                uiBothStep := 3100;
            3100:
                IF DAS_CoreSys.MachineControl.fballocatearea.fbPulloutCv.Done THEN
                    DAS_CoreSys.MachineControl.fballocatearea.M_StopStoragePulloutAction();
                    BoxReady_2nd := TRUE;
                    uiBothStep := 9999;
                END_IF

                IF DAS_CoreSys.MachineControl.fballocatearea.fbPulloutCv.Error THEN
                    DAS_CoreSys.MachineControl.fballocatearea.M_StopStoragePulloutAction();
                    uiResumeStep := 30000;
                    uiBothStep := 3000;
                    _Abort := TRUE;
                    strStatus := 'FB_RobotRegionMove_PullOutConveyor Step 30000: Feed box timeout';


                END_IF
            9999: //Wait		
        // wait reset
        END_CASE

        // Robot Abs move
        Robot.M_StartRobotAbsMove(GetBox := Get,
                                  UseClampA := UseA,
                                  UseClampB := UseB,
                                  Area := Area,
                                  ClampA_Address := Address_A,
                                  ClampB_Address := Address_B,
                                  BoxReady_1 := BoxReady_1st,
                                  BoxReady_2 := BoxReady_2nd);

        IF Robot._DI1.Done THEN
            tonTimeOut.IN := FALSE;
            uiExecutingStep := 30080;
        END_IF

        tonTimeOut.IN := TRUE;

        IF tonTimeOut.Q = TRUE THEN
            tonTimeOut.IN := FALSE;
            strStatus 	  := 'FB_RobotRegionMove_PullOutConveyor Step 30000: Robot Move timeout';
			uiResumeStep := 30000;
            _Abort := TRUE;
        END_IF
		IF robot._DI1.Error THEN
			_Abort		 := TRUE;
			strStatus	 := CONCAT('FB_RobotRegionMove_PullOutConveyor Step 30000: ',robot.ErrMsg);
			uiResumeStep := 30000;
		END_IF

    30080: // Check robot command is clear

        Robot.M_ResetRobotAbsMove(UseA, UseB);
        DAS_CoreSys.MachineControl.fballocatearea.M_StopStoragePulloutAction();

        IF NOT Robot._DI1.Done THEN
            tonTimeOut.IN := FALSE;
            uiExecutingStep := 99000; // 
        END_IF

        tonTimeOut.IN := TRUE;

        IF tonTimeOut.Q = TRUE THEN
            strStatus := 'FB_RobotRegionMove_PullOutConveyor Step 30080: Stop Robot timeout';


            _Error := TRUE;
        END_IF

    99000: // process done
        DAS_CoreSys.MachineControl.fballocatearea.M_ReleasePulloutAccess(ControlAccess := E_RoundBeltControlAccess.FanucRobot);
        Status := 'FB_RobotRegionMove_PullOutConveyor Step 99000: Process completed';
        _Executed := TRUE;
END_CASE

IF _Executed THEN
    eState := STATE_DONE;
ELSIF _Error THEN

    eState := STATE_ERROR;
ELSIF NOT Execute THEN
    eState := STATE_RESETTING;
END_IF

IF _Abort OR Abort THEN

    eSTATE := STATE_ABORTING;
END_IF
END_METHOD

METHOD  M_STATE_RESETTING
VAR_INPUT
END_VAR
// Done := false 更改到Dormant 清除確保，上位檢查到done 後可以直接下Execute

CASE uiResettingStep OF

    0:
        tonTimeOut.IN := FALSE;
        Robot.M_ResetAllCommand();
        Robot.M_ResetRobotAbsMove(TRUE, TRUE);
        uiResettingStep := 100;
        DAS_CoreSys.MachineControl.fbStorageArea.M_ResetSlides_FeedOut();
    100:

        // DAS_CoreSys.MachineControl.fbStorageArea.M_InactivePulloutConveyorInternCtrl();
        DAS_CoreSys.MachineControl.fbAllocateArea.M_ReleasePulloutAccess(ControlAccess := E_RoundBeltControlAccess.FanucRobot);
        DAS_CoreSys.MachineControl.fbAllocateArea.M_StopStoragePulloutAction();
        uiResettingStep := 9999;
    9999:
//        Done := FALSE;
//        Busy := FALSE;
        _ResetCompleted := TRUE;
END_CASE

IF _ResetCompleted THEN
    eSTATE := STATE_DORMANT;
END_IF
END_METHOD

END_FUNCTION_BLOCK

// ---- Library/20_MachineUnits/22_AllocateArea/Service/FB_AllocateRobotNeedlingMove.TcPOU
FUNCTION_BLOCK FB_AllocateRobotNeedlingMove EXTENDS FB_ActionBasic
VAR_INPUT
    xExecute      : BOOL;
    xAbort        : BOOL;
    TimeOut  : LREAL := 30; // Unit : s
	MovingInfo	: ST_AllocateRobotNeedlingMoveInfo;
END_VAR
VAR_OUTPUT
    xAborted : BOOL;
    iErrorID : INT;
    ErrorMsg : T_MaxString;
END_VAR
VAR
    StateBehavior   : CBML.ETrigATo;
    uiCyclicStep    : UINT := 0;
    uiIndexLoop     : UINT;
	Coordinate		:st_Coordinate;
	fbExecuteEdgeDetect :FB_EdgeDetect;
END_VAR

THIS^.IBehaviourModel := StateBehavior;
StateBehavior(xExecute := xExecute,
              xAbort := xAbort OR fbExecuteEdgeDetect.xFallingEdge,
              udiTimeOut := LREAL_TO_UDINT( TimeOut*1000000),
              xDone => xDone,
              xBusy => xBusy,
              xError => xError,			  
              xAborted => xAborted);			  

			  
//Make sure that C# turns off execute to shut down the service
fbExecuteEdgeDetect(xInput :=xExecute);

//Error Msg
iErrorID := StateBehavior._model.iErrorID;
ErrorMsg := M_GetErrorMsg(xErrorID := iErrorID);

METHOD CleanupAction
VAR_INPUT
    xAbortProposed : BOOL;
    iErrorIDProposed: INT;
END_VAR
VAR_OUTPUT
    xComplete : BOOL := TRUE;
    xAbort: BOOL := xAbortProposed;
 	iErrorID : INT := iErrorIDProposed;
END_VAR
uiCyclicStep := 0;
END_METHOD

METHOD CyclicAction
VAR_INPUT
    itfTimingController : CBML.ITimingController;
END_VAR
VAR_OUTPUT
    xComplete : BOOL := TRUE;
    iErrorID : INT := 0;
END_VAR
VAR_INST
	
END_VAR

VAR
		bAxesCheck 		: BOOL;
	
	
END_VAR
xComplete := FALSE;

	IF arAxisCtrl_gb[AxisNo.Allocate_X].Admin.Axis.Status.Error OR
		arAxisCtrl_gb[AxisNo.Allocate_Y].Admin.Axis.Status.Error THEN
		iErrorID :=3;
	END_IF

CASE uiCyclicStep OF
    0:
		
			uiCyclicStep:=100;
		
		
	100:
			arAxisCtrl_gb[AxisNo.Allocate_X].PosMode.Position:=Coordinate.X;
			arAxisCtrl_gb[AxisNo.Allocate_Y].PosMode.Position:=Coordinate.Y;	
		
			IF arAxisCtrl_gb[AxisNo.Allocate_X].Admin.Axis.Status.Moving OR
			   arAxisCtrl_gb[AxisNo.Allocate_Y].Admin.Axis.Status.Moving OR
			   arAxisStatus_gb[AxisNo.Allocate_X].Admin._OpModeAck=E_AXIS_MODE.ModePosAbs OR
			   arAxisStatus_gb[AxisNo.Allocate_y].Admin._OpModeAck=E_AXIS_MODE.ModePosAbs THEN
			   uiCyclicStep:=200;
			END_IF
			
	200:
			bAxesCheck := TRUE;

		bAxesCheck := bAxesCheck AND	 arAxisStatus_gb[AxisNo.Allocate_x].Admin.CmdDone ;
		bAxesCheck := bAxesCheck AND	 arAxisStatus_gb[AxisNo.Allocate_y].Admin.CmdDone ;	
	
		IF bAxesCheck THEN
			 uiCyclicStep:=600;
		END_IF
	600:
		
		xComplete := TRUE;
END_CASE
END_METHOD

METHOD ExitAction
VAR_INPUT
    xAfterCleanup : BOOL;
    xInCopyCode : BOOL;
END_VAR
END_METHOD

METHOD PRIVATE M_CheckCommand : BOOL
VAR_INPUT
END_VAR
VAR_OUTPUT
	iErrorID	 : INT :=0 ;
END_VAR
VAR
	
END_VAR
IF MovingInfo.Box<0 OR MovingInfo.Box >1 OR MovingInfo.Clip<0 OR MovingInfo.Clip>3 OR MovingInfo.NeedleLocation<0 OR MovingInfo.NeedleLocation>49 THEN
	iErrorID :=2;
	M_CheckCommand := FALSE;
	RETURN;
END_IF

IF MovingInfo.Area = 'T' THEN
		
	FUN_GetNeedleCoordinates(uiLocation :=1 ,
							 uiBox:=MovingInfo.Box,
							 uiClip:=MovingInfo.Clip,
							 uiNeedleLocation:=MovingInfo.NeedleLocation,
							 NeedleCoordinate=>Coordinate);
	IF MovingInfo.Box = 1 AND (MovingInfo.Clip = 2 OR MovingInfo.Clip = 3) THEN
		M_CheckCommand := FALSE;
		iErrorID :=2;
		RETURN;
	END_IF
	IF MovingInfo.Box = 2 AND (MovingInfo.Clip = 0 OR MovingInfo.Clip = 1) THEN
		M_CheckCommand :=FALSE;
		iErrorID :=2;
		RETURN;
	END_IF
	
ELSIF 	

	MovingInfo.Area = 'Q' THEN
	FUN_GetNeedleCoordinates(uiLocation :=0 ,
							 uiBox:=MovingInfo.Box,
							 uiClip:=MovingInfo.Clip,
							 uiNeedleLocation:=MovingInfo.NeedleLocation,
							 NeedleCoordinate=>Coordinate);
	

ELSE
	iErrorID :=2;
	M_CheckCommand := FALSE;
	RETURN;
END_IF

M_CheckCommand:=TRUE;
END_METHOD

METHOD M_GetErrorMsg : T_MaxString
VAR_INPUT
	xErrorID: INT;
END_VAR

VAR
	
END_VAR
CASE xErrorID OF
	0:
		M_GetErrorMsg := 'No Error';
	1:
		M_GetErrorMsg := 'FB_AllocateRobotNeedlingMove ErrorID 1: Action time out';
	2:
		M_GetErrorMsg := 'FB_AllocateRobotNeedlingMove ErrorID 2: Wrong command';
	3:
		M_GetErrorMsg := 'FB_AllocateRobotNeedlingMove ErrorID 3: Servo axis error';
//	4:
//		M_GetErrorMsg := 'Axis roundbelt not ready has Error';
//	5:
//		M_GetErrorMsg := 'Cylinder not ready has Error';
//	6:
//		M_GetErrorMsg := 'Axis RoundBelt has Error';
//	7:
//		M_GetErrorMsg := 'ChargeZone_Plug has Error';
//	8:
//		M_GetErrorMsg := 'TransmitCVZone_Plug has Error';
//	9:
//		M_GetErrorMsg := 'WorkZone_Plug has Error';
//	10:
//		M_GetErrorMsg := 'WorkZone_Press has Error';
END_CASE
END_METHOD

METHOD PRIVATE M_ResetAxes : BOOL
VAR_INPUT
END_VAR
VAR
	bAxesCheck :BOOL;
END_VAR
		bAxesCheck :=TRUE;
		IF arAxisCtrl_gb[AxisNo.Allocate_X].Admin.Axis.Status.Error THEN
			arAxisCtrl_gb[AxisNo.Allocate_X].Admin.ClearError:=TRUE;			
			ELSE
			arAxisCtrl_gb[AxisNo.Allocate_X].Admin.ClearError:=FALSE;	
		END_IF
		IF arAxisCtrl_gb[AxisNo.Allocate_Y].Admin.Axis.Status.Error THEN
			arAxisCtrl_gb[AxisNo.Allocate_Y].Admin.ClearError:=TRUE;			
			ELSE
			arAxisCtrl_gb[AxisNo.Allocate_Y].Admin.ClearError:=FALSE;	
		END_IF
		bAxesCheck := bAxesCheck AND NOT arAxisCtrl_gb[AxisNo.Allocate_X].Admin.ClearError ;
		bAxesCheck := bAxesCheck AND NOT arAxisCtrl_gb[AxisNo.Allocate_X].Admin.ClearError ;
		
		M_ResetAxes := bAxesCheck;
END_METHOD

METHOD ResetAction
VAR_OUTPUT
    xComplete : BOOL := TRUE;
END_VAR
uiCyclicStep := 0;
END_METHOD

METHOD StartAction
VAR_OUTPUT
    xComplete : BOOL := TRUE;
	iErrorID : INT := 0;
END_VAR
xComplete := FALSE;
uiCyclicStep := 0;

IF M_CheckCommand(iErrorID=>iErrorID) AND M_ResetAxes() THEN
	xComplete := TRUE;
END_IF
END_METHOD

END_FUNCTION_BLOCK

// ---- Library/20_MachineUnits/21_StorageArea/FB_StorageArea.TcPOU
FUNCTION_BLOCK FB_StorageArea EXTENDS FB_ModeBase_V2 IMPLEMENTS I_UnitState
VAR_INPUT
    FanucRobot : REFERENCE TO FB_FanucRobot_Basic_V2;
    Service    : REFERENCE TO ST_StorageService;

    Cylinder : REFERENCE TO UNI_CylinderList;
    Motor    : REFERENCE TO UNI_MotorList;

    Input            : REFERENCE TO ST_InputTable;
    OutPut           : REFERENCE TO ST_OutputTable;
    Reset            : REFERENCE TO BOOL;
	Stop :  REFERENCE TO BOOL;
	bStopMem :  REFERENCE TO BOOL;
    WheelhouseSensor : REFERENCE TO UNI_HMI_WheelHouseInput;
    CurrentData      : ST_SetupPara;
END_VAR
VAR_OUTPUT
	RobotResetCMD :BOOL;
	Homed : BOOL;
END_VAR
VAR
	Abort	:BOOL;

	// 連動暫停 - 任一 Service 錯誤時暫停所有其他 Service
	_bAnyServiceError : BOOL;

    // Service
    //fbFeedInEmptyBoxWithRobot           : FB_FeedInEmptyBoxWithRobot;
	fbFeedInEmptyBoxWithRobot           : FB_FeedInEmptyBoxWithRobot_V4;			//Edited by Gamin in 2025//11/24
    //fbReloadRoundBeltBoxWithRobot       : FB_ReloadRoundBeltBoxWithRobot;
	fbReloadRoundBeltBoxWithRobot       : FB_ReloadRoundBeltBoxWithRobot_V2;		//Edited by Gamin in 2025//11/24
    fbRobotRegionMove_AllocatedConveyor : FB_RobotRegionMove_AllocatedConveyor;
    fbRobotRegionMove_BufferArea        : FB_RobotRegionMove_BufferArea;
    //fbRobotRegionMove_FeedInConveyor    : FB_RobotRegionMove_FeedInConveyor;
	fbRobotRegionMove_FeedInConveyor    : FB_RobotRegionMove_FeedInConveyor_V2;		//Edited by Gamin in 2025//11/24
    fbRobotRegionMove_PullOutConveyor   : FB_RobotRegionMove_PullOutConveyor;
    fbRobotRegionMove_RoundBelt         : FB_RobotRegionMove_RoundBelt;
    //fbRobotAbsMove                      : FB_RobotAbsMove;
	fbRobotAbsMove                      : FB_RobotAbsMove_V2;
    //fbWareHouseWithRobotMove            : FB_WareHouseWithRobotMove;
    fbWareHouseWithRobotMove             : FB_WareHouseWithRobotMove_V3;		//Edited by Gamin in 2025//11/24
	fbFeedInRoundBeltBoxToWareHouse 	 : FB_FeedInRoundBeltBoxToWareHouse;
	fbWareHouseInnerPickToRoundBelt 	 : FB_WareHouseInnerPickToRoundBelt;
	fbWareHouseInnerPickToRoundBeltBatch : FB_WareHouseInnerPickToRoundBeltBatch;
	fbFeedInRoundBeltBoxBatch			 : FB_FeedInRoundBeltBoxBatch;
	fbRobotSelfHoming					 : FB_RobotSelfHoming;
	
	fbStorageHoming 					: FB_StorageHoming;
	//UpCV
    _fbDaimeterMovement   			: FB_DiameterMovement; //UpCV Internal use
    fbUpperFeedInConveyor 			: FB_UpperFeedInConveyor;
	bUpperCV_ServiceDone			: BOOL;					// 偵測上層輸送帶是否做完
	fbAddBoxes                      : FB_AddBoxes_v2;
	fbBoxSupplyCtrl					: FB_BoxSupplyCtrl_v1;
    RackState                       : E_RackState;
    
    // Pullout
    fbPullOutConveyorAction         : FB_PullOutConveyorAction;
    AutoPullout_Ctrl                : ST_AutoPullOutConveyorCommand;
    AutoPullout_Status              : ST_AutoPullOutConveyorSatus;
    AutoPullout_Info                : ST_PullOutConveyorInfo;
    bPulloutConveyorInternCtrl      : BOOL := FALSE;
    AutoMode_PulloutConveyor_Intern : ST_AutoPullOutConveyor; // Pullout conveyor inter
    

    // Robot abs move
    RobotAbsMoveAuto_Ctrl   : st_RobotAbsMove_Ctrl;
    RobotAbsMoveAuto_Status : st_RobotAbsMove_Status;
    RobotAbsMoveAuto_Info   : st_AutoSixAxisAbsMoveParameter;
    // Warehouse
	fbWarehouse           : FB_WareHouse;
    //========= Auto Mode Robot Warehouse Move =================
    RobotWarehouseMoveAuto_Ctrl   : st_RobotWarehouseMove_Ctrl;
    RobotWarehouseMoveAuto_Status : st_RobotWarehouseMove_Status;

    _RobotWarehouseMoveAuto_Ctrl   : st_RobotWarehouseMove_Ctrl;
    _RobotWarehouseMoveAuto_Status : st_RobotWarehouseMove_Status;

    RobotWarehouseMoveAuto_internal_Ctrl   : st_RobotWarehouseMove_Ctrl;
    RobotWarehouseMoveAuto_internal_Status : st_RobotWarehouseMove_Status;
    bWarehouseMoveInternalAccess           : BOOL := FALSE;
	// Storage homing
	StorageHoming_Execute : BOOL;
	StorageHoming_Reset : BOOL;
	StorageHoming_Abort : BOOL;
	StorageHoming_Busy : BOOL;
	StorageHoming_Done : BOOL;
	StorageHoming_Error : BOOL;
	
	// Reboot Modbus devices
	fbRebootModbusDevice		: FB_RebootModbusDevice;
END_VAR

SUPER^();

IF __ISVALIDREF(PackTag) THEN
    eModeCommand := PackTag.Command.UnitMode;
    eStateCommand := PackTag.Command.CntrlCmd;
ELSE
    RETURN;
END_IF

ACTION A00_Service:
// ============================================================================
// 連動暫停邏輯 - 任一 Service 錯誤時，暫停所有其他 Service
// ============================================================================
//_bAnyServiceError :=
//	service.AutoMode_FeedInEmptyBoxWithRobot.Status.Error OR
//	service.AutoMode_RobotRegionMove_BufferArea.Status.Error OR
//	service.AutoMode_UpperFeedInConveyor.Status.Error OR
//	service.AutoMode_AddBoxes.Status.Error OR
//	service.AutoMode_RobotRegionMove_FeedInConveyor.Status.Error OR
//	service.AutoMode_RobotRegionMove_AllocatedConveyor.Status.Error OR
//	service.AutoMode_RobotRegionMove_PullOutConveyor.Status.Error OR
//	service.AutoMode_RobotAbsMove.HandShake.Error OR
//	service.AutoMode_RobotRegionMove_RoundBelt.Status.Error OR
//	service.AutoMode_ReloadRoundBeltBoxWithRobot.Status.Error OR
//	service.AutoMode_WarehouseMotoWithRobotMove.HandShake.Error OR
//	AutoPullout_Status.Error;

fbFeedInEmptyBoxWithRobot(Execute    := service.AutoMode_FeedInEmptyBoxWithRobot.Command.Execute,
                          Abort      := service.AutoMode_FeedInEmptyBoxWithRobot.Command.Abort OR THIS^.Abort OR _bAnyServiceError,
                          Reset      := service.AutoMode_FeedInEmptyBoxWithRobot.Command.Reset,
                          ObjectName := 'FeedInEmptyBox with robot',
                          Busy       => service.AutoMode_FeedInEmptyBoxWithRobot.Status.Busy,
                          Done       => service.AutoMode_FeedInEmptyBoxWithRobot.Status.Done,
                          Aborted    =>,
                          Error      => service.AutoMode_FeedInEmptyBoxWithRobot.Status.Error,
                          ErrorID    =>,
                          Status     => service.AutoMode_FeedInEmptyBoxWithRobot.Status.Status,
                          UniqueErrorCode   =>,
                          Robot      := FanucRobot,
                          WareHouse  := fbWarehouse,
                          Input      := Input,
                          DiffSizeCV := Motor.List.TransmitDifferentSideCV,
						  SameSizeCV := Motor.List.TransmitSameSideCV,
                          Info := Service.AutoMode_FeedInEmptyBoxWithRobot.Info,
                          Pause := bStopMem,
                          Stop := bStopMem,
						  AClampMoveDone=>service.AutoMode_FeedInEmptyBoxWithRobot.AClampMoveDone,
						  BClampMoveDone=>service.AutoMode_FeedInEmptyBoxWithRobot.BClampMoveDone);

fbRobotRegionMove_BufferArea(Execute	:= Service.AutoMode_RobotRegionMove_BufferArea.Command.Execute,
                             Abort 		:= Service.AutoMode_RobotRegionMove_BufferArea.Command.Abort OR THIS^.Abort OR _bAnyServiceError,
                             Reset 		:= Service.AutoMode_RobotRegionMove_BufferArea.Command.Reset,
                             ObjectName	:= 'RobotRegionMove_BufferArea',
                             Busy    => Service.AutoMode_RobotRegionMove_BufferArea.Status.Busy,
                             Done    => Service.AutoMode_RobotRegionMove_BufferArea.Status.Done,
                             Aborted =>,
                             Error   => Service.AutoMode_RobotRegionMove_BufferArea.Status.Error,
                             ErrorID =>,
                             Status  => Service.AutoMode_RobotRegionMove_BufferArea.Status.Status,
							 UniqueErrorCode	=>,
                             Robot 	:= FanucRobot,
                             Info 	:= Service.AutoMode_RobotRegionMove_BufferArea.Info,
                             Stop 	:= bStopMem);

fbPullOutConveyorAction(Execute          := (*AutoPullout_Ctrl.Execute*) ,
                        Abort            := AutoPullout_Ctrl.Abort OR THIS^.Abort OR _bAnyServiceError,
                        Reset            := AutoPullout_Ctrl.Reset,
                        ObjectName       := 'fbPullOutConveyorAction',
                        Busy             => AutoPullout_Status.Busy,
                        Done             => AutoPullout_Status.Done,
                        Aborted          =>,
                        Error            => AutoPullout_Status.Error,
                        ErrorID          =>,
                        Status           => AutoPullout_Status.Status,
                        UniqueErrorCode  =>,
                        FixCylinderA1    := Cylinder.List.fbPullOutCV_AsidePress1,
                        FixCylinderA2    := Cylinder.List.fbPullOutCV_AsidePress2,
                        FixCylinderB1    := Cylinder.List.fbPullOutCV_BsidePress1,
                        FixCylinderB2    := Cylinder.List.fbPullOutCV_BsidePress2,
                        BarrierCylinderA := Cylinder.List.fbPullOutCV_AsideBlock,
                        BarrierCylinderB := Cylinder.List.fbPullOutCV_BsideBlock,
                        ConveyorMotorA   := Motor.List.PullOutCV_A,
                        ConveyorMotorB   := Motor.List.PullOutCV_B,
                        INPUT            := INPUT,
                        PullOutInfo      := AutoPullout_Info);

fbUpperFeedInConveyor(Execute             := Service.AutoMode_UpperFeedInConveyor.Command.Execute,
                      Abort               := Service.AutoMode_UpperFeedInConveyor.Command.Abort OR THIS^.Abort OR _bAnyServiceError,
                      Reset               := Service.AutoMode_UpperFeedInConveyor.Command.Reset,
                      ObjectName          := 'Storage_UpperFeedInConveyor',
                      Busy                => Service.AutoMode_UpperFeedInConveyor.Status.Busy,
                      Done                => Service.AutoMode_UpperFeedInConveyor.Status.Done,
                      Aborted             =>,
                      Error               => Service.AutoMode_UpperFeedInConveyor.Status.Error,
                      ErrorID             =>,
                      Status              =>,
                      UniqueErrorCode     =>,
                      _fbDiameterMovement := THIS^._fbDaimeterMovement,
                      Cylinder            := Cylinder,
                      Motor               := Motor,
                      Input               := Input,
                      OutPut              := OutPut,
                      Info                := Service.AutoMode_UpperFeedInConveyor.Info,
                      AddingBox           :=,
                      FeedBack            => Service.AutoMode_UpperFeedInConveyor.FeedBack,
					  _bForceUpperCV_Use  =>	,
					  Pause 			  := bStopMem,
					  RobotService_CheckUPCVServicedone =>bUpperCV_ServiceDone);

_fbDaimeterMovement(Execute         :=,
                    Abort           := _bAnyServiceError,
                    Reset           :=,
                    ObjectName      :=,
                    Busy            =>,
                    Done            =>,
                    Aborted         =>,
                    Error           =>,
                    ErrorID         =>,
                    Status          =>,
                    UniqueErrorCode =>,
                    bContinue       :=,
                    Cylinder        := Cylinder,
                    PickDone        =>);

fbWarehouse(Motors           := Motor,
            WheelhouseSensor := WheelhouseSensor);

fbAddBoxes(Execute                   := Service.AutoMode_AddBoxes.Command.Execute,
           Abort                     := Service.AutoMode_AddBoxes.Command.Abort OR THIS^.Abort OR _bAnyServiceError,
           Reset                     := Service.AutoMode_AddBoxes.Command.Reset,
           ObjectName                := 'Storage_AddBoxes',
           Busy                      => Service.AutoMode_AddBoxes.Status.Busy,
           Done                      => Service.AutoMode_AddBoxes.Status.Done,
           Aborted                   =>,
           Error                     => Service.AutoMode_AddBoxes.Status.Error,
           ErrorID                   =>,
           Status                    =>,
           UniqueErrorCode           =>,
           Cylinder                  := Cylinder,
           Motor                     := Motor,
           Input                     := Input,
           OutPut                    := OutPut,
           CurrentData               := CurrentData,
           ERackState                := RackState,
           bClearInterventionRequest :=,
           InterventionRequest       => Service.AutoMode_AddBoxes.Status.InterventionRequest,
           FeedingBoxes              => Service.AutoMode_AddBoxes.Status.FeedingBoxes,
			_bForceUpperCV_Use 		:= fbUpperFeedInConveyor._bForceUpperCV_Use);

fbBoxSupplyCtrl(Execute           := TRUE,
                Abort             :=THIS^.Abort OR _bAnyServiceError,
                Reset             :=reset,
                ObjectName        :=,
                Busy              =>,
                Done              =>,
                Aborted           =>,
                Error             =>,
                ErrorID           =>,
                Status            =>,
                UniqueErrorCode   =>,
                Cylinder          := Cylinder,
                Motor             := Motor,
                CurrentData       := CurrentData,
                Input             := Input,
                Output            := OutPut,
                StroageRegionMode := eModeCurrent,
                bAddsBoxRequest   := Service.AutoMode_AddBoxes.Status.InterventionRequest,
                AddBoxes_Status   := Service.AutoMode_AddBoxes.Status,
                AddBoxes_Ctrl     := Service.AutoMode_AddBoxes.Command,
				AxisRackMotorBTNHomeRequest=>,
                RackState         => RackState,
				fbstorageHome := fbStorageHoming);

fbRobotRegionMove_FeedInConveyor(Execute 	:= Service.AutoMode_RobotRegionMove_FeedInConveyor.Command.Execute,
                                 Abort 		:= Service.AutoMode_RobotRegionMove_FeedInConveyor.Command.Abort OR THIS^.Abort OR _bAnyServiceError,
                                 Reset      := Service.AutoMode_RobotRegionMove_FeedInConveyor.Command.Reset,
                                 ObjectName := 'Storage Robot FeedIn CV',
                                 Busy       => Service.AutoMode_RobotRegionMove_FeedInConveyor.Status.Busy,
                                 Done 		=> Service.AutoMode_RobotRegionMove_FeedInConveyor.Status.Done,
                                 Aborted	=>,
                                 Error   	=> Service.AutoMode_RobotRegionMove_FeedInConveyor.Status.Error,
                                 ErrorID 	=>,
                                 Status  	=> Service.AutoMode_RobotRegionMove_FeedInConveyor.Status.Status,
                                 UniqueErrorCode =>,
                                 Robot           := FanucRobot,
                                 LowerConveyor   := Motor.List.LowCV,
                                 Input           := Input,
                                 //								 F1SensorOfUpperConveyor :=Input.bUpCV_BoxArrived_Sensor,
                                 //								 Input.bUpCV_Block1Detect_Sensor := Input.bUpCV_Block1Detect_Sensor ,
                                 Info := Service.AutoMode_RobotRegionMove_FeedInConveyor.Info,
                                 Stop :=bStopMem,
								 bCheckUpperCV_ServiceDone :=	bUpperCV_ServiceDone);

fbRobotRegionMove_AllocatedConveyor(Execute 	:= Service.AutoMode_RobotRegionMove_AllocatedConveyor.Command.Execute,
                                    Abort 		:= Service.AutoMode_RobotRegionMove_AllocatedConveyor.Command.Abort OR THIS^.Abort OR _bAnyServiceError,
                                    Reset  		:= Service.AutoMode_RobotRegionMove_AllocatedConveyor.Command.Reset,
                                    ObjectName 	:= ' Storage Robot Transmit CV',
                                    Busy       	=> Service.AutoMode_RobotRegionMove_AllocatedConveyor.Status.Busy,
                                    Done 		=> Service.AutoMode_RobotRegionMove_AllocatedConveyor.Status.Done,
                                    Aborted 	=>,
                                    Error   	=> Service.AutoMode_RobotRegionMove_AllocatedConveyor.Status.Error,
                                    ErrorID 	=>,
                                    Status  	=> Service.AutoMode_RobotRegionMove_AllocatedConveyor.Status.Status,
                                    UniqueErrorCode =>,
                                    Robot           := FanucRobot,
                                    DifferenceCV    := Motor.List.TransmitDifferentSideCV,
                                    SamesizeCV      := Motor.List.TransmitSameSideCV,
                                    cylinder        := Cylinder,
                                    //	SameSizeFullSensor:= , 
                                    Input := Input,
                                    Info := service.AutoMode_RobotRegionMove_AllocatedConveyor.Info,
                                    Stop :=bStopMem);


fbRobotRegionMove_PullOutConveyor(Execute 	:=Service.AutoMode_RobotRegionMove_PullOutConveyor.Command.Execute,
                                  Abort 	:=Service.AutoMode_RobotRegionMove_PullOutConveyor.Command.Abort OR THIS^.Abort OR _bAnyServiceError,
                                  Reset     := Service.AutoMode_RobotRegionMove_PullOutConveyor.Command.Reset,
                                  ObjectName:= 'Storage Robot PulloutCV',
                                  Busy      => Service.AutoMode_RobotRegionMove_PullOutConveyor.Status.Busy,
                                  Done 		=> Service.AutoMode_RobotRegionMove_PullOutConveyor.Status.Done,
                                  Aborted 	=>,
                                  Error   	=> Service.AutoMode_RobotRegionMove_PullOutConveyor.Status.Error,
                                  ErrorID 	=>,
                                  Status  	=> Service.AutoMode_RobotRegionMove_PullOutConveyor.Status.Status,
                                  UniqueErrorCode =>,
                                  Robot           := FanucRobot,
                                  PullOutConveyor := fbPullOutConveyorAction,
                                  Info := Service.AutoMode_RobotRegionMove_PullOutConveyor.Info,
                                  Stop :=bStopMem);

fbRobotAbsMove(Execute         := Service.AutoMode_RobotAbsMove.HandShake.Execute,
               Abort           := THIS^.Abort OR _bAnyServiceError,
               Reset           := Service.AutoMode_RobotAbsMove.HandShake.Reset,
               ObjectName      := 'Storage robot abs move',
               Busy            => Service.AutoMode_RobotAbsMove.HandShake.Busy,
               Done            => Service.AutoMode_RobotAbsMove.HandShake.Done,
               Aborted         =>,
               Error           => Service.AutoMode_RobotAbsMove.HandShake.Error,
               ErrorID         =>,
               Status          =>,
               UniqueErrorCode =>,
               Robot           := FanucRobot,
               LowerConveyor   := Motor.List.LowCV,
               Info            := Service.AutoMode_RobotAbsMove,
               Input 		:= Input,
               Stop :=bStopMem,
			   	Output:=OutPut,
				Cylinder:= Cylinder,
				AClampMoveDone=>Service.AutoMode_RobotAbsMove.AClampMoveDone,
				BClampMoveDone=>Service.AutoMode_RobotAbsMove.BClampMoveDone,
				bCheckUpperCV_ServiceDone :=bUpperCV_ServiceDone);

fbRobotRegionMove_RoundBelt(Execute := Service.AutoMode_RobotRegionMove_RoundBelt.Command.Execute,
                            Abort   := THIS^.Abort OR _bAnyServiceError,
                            Reset   := Service.AutoMode_RobotRegionMove_RoundBelt.Command.Reset,
                            ObjectName:= 'Storage robot  RegionMove roundbelt',
                            Busy    => Service.AutoMode_RobotRegionMove_RoundBelt.Status.Busy,
                            Done    => Service.AutoMode_RobotRegionMove_RoundBelt.Status.Done,
                            Aborted =>,
                            Error   => Service.AutoMode_RobotRegionMove_RoundBelt.Status.Error,
                            ErrorID =>,
                            Status 	=> Service.AutoMode_RobotRegionMove_RoundBelt.Status.Status,
                            UniqueErrorCode =>,
                            Robot 		:= FanucRobot,
                            RoundBelt 	:= DAS_CoreSys.MachineControl.fbAllocateArea.RoundBeltControl,
							Input 		:= Input,
                            Info 		:= Service.AutoMode_RobotRegionMove_RoundBelt.Info,
                            Stop 		:=bStopMem);

fbReloadRoundBeltBoxWithRobot(Execute	:= Service.AutoMode_ReloadRoundBeltBoxWithRobot.Command.Execute,
                              Abort 	:= THIS^.Abort OR _bAnyServiceError,
                              Reset 	:= Service.AutoMode_ReloadRoundBeltBoxWithRobot.Command.Reset,
                              ObjectName:= 'Storage robot reload roundbelt',
                              Busy    => Service.AutoMode_ReloadRoundBeltBoxWithRobot.Status.Busy,
                              Done    => Service.AutoMode_ReloadRoundBeltBoxWithRobot.Status.Done,
                              Aborted =>,
                              Error   => Service.AutoMode_ReloadRoundBeltBoxWithRobot.Status.Error,
                              ErrorID =>,
                              Status  => Service.AutoMode_ReloadRoundBeltBoxWithRobot.Status.Status,
                              UniqueErrorCode =>,
                              Robot 	:= FanucRobot,
                              RoundBelt := DAS_CoreSys.MachineControl.fbAllocateArea.RoundBeltControl,
                              WareHouse := fbWarehouse,
                              Input 	:= Input,
                              Info 		:= Service.AutoMode_ReloadRoundBeltBoxWithRobot.Info,
                              Stop 		:= bStopMem,
							  AClampMoveDone=>Service.AutoMode_ReloadRoundBeltBoxWithRobot.AClampMoveDone,
							  BClampMoveDone=>Service.AutoMode_ReloadRoundBeltBoxWithRobot.BClampMoveDone);
							  
fbWareHouseInnerPickToRoundBelt(Execute	:= Service.AutoMode_WareHouseInnerPickToRoundBelt.Command.Execute,
                                Abort 	:= THIS^.Abort OR _bAnyServiceError,
                                Reset 	:= Service.AutoMode_WareHouseInnerPickToRoundBelt.Command.Reset,
                                ObjectName:= 'Warehouse inner pick to roundbelt',
                                Busy    => Service.AutoMode_WareHouseInnerPickToRoundBelt.Status.Busy,
                                Done    => Service.AutoMode_WareHouseInnerPickToRoundBelt.Status.Done,
                                Aborted =>,
                                Error   => Service.AutoMode_WareHouseInnerPickToRoundBelt.Status.Error,
                                ErrorID =>,
                                Status  => Service.AutoMode_WareHouseInnerPickToRoundBelt.Status.Status,
                                UniqueErrorCode =>,
                                Robot 	:= FanucRobot,
                                RoundBelt := DAS_CoreSys.MachineControl.fbAllocateArea.RoundBeltControl,
                                WareHouse := fbWarehouse,
                                Input 	:= Input,
                                Info 	:= Service.AutoMode_WareHouseInnerPickToRoundBelt.Info,
                                Stop 	:= bStopMem,
                                ReadComplete := Service.AutoMode_WareHouseInnerPickToRoundBelt.ReadComplete,
                                ActionRecords=>Service.AutoMode_WareHouseInnerPickToRoundBelt.ActionRecords,
                                ActionIndex=>Service.AutoMode_WareHouseInnerPickToRoundBelt.ActionIndex,
                                FeedBack=>Service.AutoMode_WareHouseInnerPickToRoundBelt.FeedBack);
fbWareHouseInnerPickToRoundBeltBatch(
                                Abort 	:= THIS^.Abort OR _bAnyServiceError,
                                ObjectName:= 'Warehouse inner pick batch',
                                Robot 	:= FanucRobot,
                                RoundBelt := DAS_CoreSys.MachineControl.fbAllocateArea.RoundBeltControl,
                                WareHouse := fbWarehouse,
                                Input 	:= Input,
                                BatchInfo := Service.AutoMode_WareHouseInnerPickToRoundBeltBatch,
                                Stop 	:= bStopMem);
// 圓帶回倉/PullOut 批次服務
fbFeedInRoundBeltBoxBatch(
                                Abort 	:= THIS^.Abort OR _bAnyServiceError,
                                ObjectName:= 'FeedIn round belt box batch',
                                Robot 	:= FanucRobot,
                                RoundBelt := DAS_CoreSys.MachineControl.fbAllocateArea.RoundBeltControl,
                                WareHouse := fbWarehouse,
                                Input 	:= Input,
                                BatchInfo := Service.AutoMode_FeedInRoundBeltBoxBatch,
                                Stop 	:= bStopMem);
								
//============================ Auto Mode Robot Warehouse Move =============================
IF NOT bWarehouseMoveInternalAccess THEN
    _RobotWarehouseMoveAuto_Ctrl := RobotWarehouseMoveAuto_Ctrl;
    RobotWarehouseMoveAuto_Status := _RobotWarehouseMoveAuto_Status;
ELSE
    _RobotWarehouseMoveAuto_Ctrl := RobotWarehouseMoveAuto_internal_Ctrl;
    RobotWarehouseMoveAuto_internal_Status := _RobotWarehouseMoveAuto_Status;
END_IF

(*M_RobotWarehouseMove(
        bExecute  := Service.AutoMode_RobotWarehouseMove.HandShake.Execute,
        bReset    := Service.AutoMode_RobotWarehouseMove.HandShake.Reset,
        bAbort    := FALSE,
        bOccupied := FALSE,
        eMode     := E_MachineMode.Auto,
        bBusy     => Service.AutoMode_RobotWarehouseMove.HandShake.Busy,
        bDone     => Service.AutoMode_RobotWarehouseMove.HandShake.Done,
        bError    => Service.AutoMode_RobotWarehouseMove.HandShake.Error);*)
fbWareHouseWithRobotMove(
	Execute:= Service.AutoMode_WarehouseMotoWithRobotMove.HandShake.Execute,
	Abort:= THIS^.Abort OR _bAnyServiceError,
	Reset:= Service.AutoMode_WarehouseMotoWithRobotMove.HandShake.Reset,
	ObjectName:= 'storage Robot Warehouse move', 
	Busy=> Service.AutoMode_WarehouseMotoWithRobotMove.HandShake.Busy, 
	Done=> Service.AutoMode_WarehouseMotoWithRobotMove.HandShake.Done, 
	Aborted=> , 
	Error=> Service.AutoMode_WarehouseMotoWithRobotMove.HandShake.Error, 
	ErrorID=> , 
	Status=> , 
	UniqueErrorCode=> , 
	Robot:= FanucRobot, 
	WareHouse:= fbWarehouse, 
	Info:= Service.AutoMode_WarehouseMotoWithRobotMove, 
	Stop:= bStopMem,
	AClampMoveDone=> Service.AutoMode_WarehouseMotoWithRobotMove.AClampMoveDone,
	BClampMoveDone=> Service.AutoMode_WarehouseMotoWithRobotMove.BClampMoveDone,
	WarehouseStatus := WheelhouseSensor.List);
	
fbStorageHoming(
	xDone=> ,
	xBusy=> ,
	xError=> ,
	xExecute:= ,
	xAbort:= THIS^.Abort OR _bAnyServiceError,
	Cylinder:= Cylinder, 
	Motor:= Motor, 
	FanucRobot:= FanucRobot,
	Homed := Homed,
	xAborted=> , 
	iErrorID=> , 
	ErrorMsg=> , 
	RobotResetCMD=> RobotResetCMD,
	RackMotorHomeRequest=>,
	Input := Input,
	Service := Service,
	Output :=OutPut);
	
fbRebootModbusDevice(
	xDone=> Service.RebootModbusDevices.Status.Done, 
	xBusy=> Service.RebootModbusDevices.Status.Busy, 
	xError=> Service.RebootModbusDevices.Status.Error, 
	xExecute:= Service.RebootModbusDevices.Command.Execute, 
	xAbort:= Service.RebootModbusDevices.Command.Abort, 
	OutPut:= OutPut, 
	OffDelayTime:= Service.RebootModbusDevices.OffDelayTime, 
	OnDelayTime:= Service.RebootModbusDevices.OnDelayTime, 
	xAborted=> , 
	iErrorID=> , 
	ErrorMsg=> );
	
fbFeedInRoundBeltBoxToWareHouse(
	Execute:= Service.AutoMode_FeedInRoundBeltBoxToWareHouse.Command.Execute, 
	Abort:= , 
	Reset:= Service.AutoMode_FeedInRoundBeltBoxToWareHouse.Command.Reset, 
	Pause:= , 
	ObjectName:= , 
	Busy=> Service.AutoMode_FeedInRoundBeltBoxToWareHouse.Status.Busy, 
	Done=> Service.AutoMode_FeedInRoundBeltBoxToWareHouse.Status.Done, 
	Aborted=> , 
	Error=> Service.AutoMode_FeedInRoundBeltBoxToWareHouse.Status.Error, 
	Paused=> , 
	ErrorID=> , 
	Status=> Service.AutoMode_FeedInRoundBeltBoxToWareHouse.Status.Status, 
	UniqueErrorCode=> , 
	Robot:= FanucRobot, 
	RoundBelt:= DAS_CoreSys.MachineControl.fbAllocateArea.RoundBeltControl, 
	WareHouse:= fbWarehouse, 
	Input:= Input, 
	Info:= Service.AutoMode_FeedInRoundBeltBoxToWareHouse.Info, 
	Stop:= bStopMem, 
	AClampMoveDone=> Service.AutoMode_FeedInRoundBeltBoxToWareHouse.AClampMoveDone, 
	BClampMoveDone=> Service.AutoMode_FeedInRoundBeltBoxToWareHouse.BClampMoveDone);
	
fbRobotSelfHoming(
	Execute:= Service.AutoMode_RobotSelfHoming.Command.Execute, 
	Abort:= , 
	Reset:= Service.AutoMode_RobotSelfHoming.Command.Reset, 
	Pause:= bStopMem, 
	ObjectName:= 'FB_RobotSelfHoming', 
	Busy=> Service.AutoMode_RobotSelfHoming.Status.Busy, 
	Done=> Service.AutoMode_RobotSelfHoming.Status.Done, 
	Aborted=> , 
	Error=> Service.AutoMode_RobotSelfHoming.Status.Error, 
	Paused=> , 
	ErrorID=> , 
	Status=> Service.AutoMode_RobotSelfHoming.Status.Status, 
	UniqueErrorCode=> , 
	FanucRobot:= FanucRobot, 
	Input:= Input, 
	Output:= OutPut, 
	Motor:= Motor, 
	BypassFeedOutToNGCV:= Service.AutoMode_RobotSelfHoming.BypassFeedOutToNGCV);
END_ACTION

METHOD M_Aborted
Abort:=FALSE;
M_StopHoming();
M_StateComplete();
END_METHOD

METHOD M_AbortHoming
VAR_INPUT
END_VAR
StorageHoming_Abort := TRUE;
END_METHOD

METHOD M_Aborting
Abort := TRUE;
M_StateComplete();
END_METHOD

METHOD M_ActivePulloutConveyorInternCtrl : BOOL
VAR_INPUT
END_VAR
bPulloutConveyorInternCtrl := TRUE;

M_ActivePulloutConveyorInternCtrl := TRUE; // Method end
END_METHOD

METHOD M_ActivePulloutConveyorInternCtrl_1 : BOOL
VAR_INPUT
END_VAR
bPulloutConveyorInternCtrl := TRUE;

M_ActivePulloutConveyorInternCtrl_1 := TRUE; // Method end
END_METHOD

METHOD M_AutoPullOutConveyorActive : BOOL
VAR_INPUT
END_VAR
IF eModeCurrent = E_UnitMode.AUTO AND NOT bPulloutConveyorInternCtrl THEN
    // GVL -> AutoSimpleAllocate_Ctrl
    AutoPullout_Ctrl.Execute := service.AutoMode_PullOutConveyor.Command.Execute;
    AutoPullout_Ctrl.Abort   := service.AutoMode_PullOutConveyor.Command.Abort;
    AutoPullout_Ctrl.Reset   := service.AutoMode_PullOutConveyor.Command.Reset OR Reset;
	M_LoadingPullOutConveyorData();
ELSIF eModeCurrent = E_UnitMode.AUTO AND bPulloutConveyorInternCtrl THEN
    AutoPullout_Ctrl.Execute := AutoMode_PulloutConveyor_Intern.Command.Execute;
    AutoPullout_Ctrl.Abort   := AutoMode_PulloutConveyor_Intern.Command.Abort;
    AutoPullout_Ctrl.Reset   := AutoMode_PulloutConveyor_Intern.Command.Reset OR Reset;
	M_LoadingPullOutConveyorData();
ELSE
    AutoPullout_Ctrl.Execute := FALSE;
    AutoPullout_Ctrl.Abort   := FALSE;
    AutoPullout_Ctrl.Reset   := FALSE;
END_IF

// AutoSimpleAllocate_Status - > GVL
service.AutoMode_PullOutConveyor.Status.Busy := AutoPullout_Status.Busy;
service.AutoMode_PullOutConveyor.Status.Done := AutoPullout_Status.Done;
service.AutoMode_PullOutConveyor.Status.Error:= AutoPullout_Status.Error;
AutoMode_PulloutConveyor_Intern.Status.Busy := AutoPullout_Status.Busy;
AutoMode_PulloutConveyor_Intern.Status.Done:= AutoPullout_Status.Done;
AutoMode_PulloutConveyor_Intern.Status.Error:= AutoPullout_Status.Error;
END_METHOD

METHOD M_Clearing
M_StateComplete();
END_METHOD

METHOD M_Complete
M_StateComplete();
END_METHOD

METHOD M_Completing
M_StateComplete();
END_METHOD

METHOD M_Execute
CASE eModeCurrent OF
	E_UnitMode.Manual:
	
	E_UnitMode.Auto:
END_CASE
A00_Service();
//M_StateComplete();
END_METHOD

METHOD M_Held
M_StateComplete();
END_METHOD

METHOD M_Holding
//fbRobotRegionMove_BufferArea.Stop := TRUE;
M_StateComplete();
END_METHOD

METHOD M_Idle
M_StateComplete();
END_METHOD

METHOD M_InactivePulloutConveyorInternCtrl : BOOL
VAR_INPUT
END_VAR
bPulloutConveyorInternCtrl := FALSE;

M_InactivePulloutConveyorInternCtrl := TRUE; // Method end
END_METHOD

METHOD PRIVATE M_LoadingPullOutConveyorData : BOOL
VAR_INPUT
END_VAR
IF eModeCurrent = E_UnitMode.Manual AND NOT bPulloutConveyorInternCtrl THEN
    AutoPullout_Info := Service.AutoMode_PullOutConveyor .PullOutConveyorInfo;
ELSIF eModeCurrent = E_UnitMode.Auto AND bPulloutConveyorInternCtrl THEN
    AutoPullout_Info := AutoMode_PulloutConveyor_Intern.PullOutConveyorInfo;
END_IF

M_LoadingPullOutConveyorData := TRUE; // Method end
END_METHOD

METHOD M_ResetSlideA_FeedIn : BOOL
VAR_INPUT
END_VAR
AutoMode_PulloutConveyor_Intern.Command.Execute := FALSE;

M_ResetSlideA_FeedIn := FALSE;
END_METHOD

METHOD M_ResetSlideB_FeedIn : BOOL
VAR_INPUT
END_VAR
AutoMode_PulloutConveyor_Intern.Command.Execute := FALSE;

M_ResetSlideB_FeedIn := FALSE;
END_METHOD

METHOD M_ResetSlides_FeedOut : BOOL
VAR_INPUT
END_VAR
AutoMode_PulloutConveyor_Intern.Command.Execute := FALSE;

M_ResetSlides_FeedOut := FALSE;
END_METHOD

METHOD M_Resetting
M_StateComplete();
END_METHOD

METHOD M_RobotWarehouseMove : BOOL
VAR_INPUT
	bExecute			: BOOL;
	bReset				: BOOL;
	bAbort				: BOOL;
	bOccupied			: BOOL;
	eMode				: E_MachineMode;
END_VAR

VAR_OUTPUT
	bBusy				: BOOL;
	bDone				: BOOL;
	bError				: BOOL;
END_VAR
CASE eMode OF
	E_MachineMode.MANUAL:
//		RobotWarehouseMoveManual_Ctrl.bExecute := bExecute;
//		RobotWarehouseMoveManual_Ctrl.bReset := bReset;
//		RobotWarehouseMoveManual_Ctrl.bAbort := E_Stop;
//		RobotWarehouseMoveManual_Ctrl.bOccupied := bOccupied;
		
//		bBusy := RobotWarehouseMoveManual_Status.bBusy;
//		bDone := RobotWarehouseMoveManual_Status.bDone;
//		bError := RobotWarehouseMoveManual_Status.bError;
		
	E_MachineMode.AUTO:
//		RobotWarehouseMoveAuto_Ctrl.bExecute := bExecute;
//		RobotWarehouseMoveAuto_Ctrl.bReset := bReset;
//		RobotWarehouseMoveAuto_Ctrl.bAbort := E_Stop;
//		RobotWarehouseMoveAuto_Ctrl.bOccupied := bOccupied;
		
//		bBusy := RobotWarehouseMoveAuto_Status.bBusy;
//		bDone := RobotWarehouseMoveAuto_Status.bDone;
//		bError := RobotWarehouseMoveAuto_Status.bError;
END_CASE
END_METHOD

METHOD M_RobotWarehouseMove_1 : BOOL
VAR_INPUT
	bExecute			: BOOL;
	bReset				: BOOL;
	bAbort				: BOOL;
	bOccupied			: BOOL;
	eMode				: E_MachineMode;
END_VAR

VAR_OUTPUT
	bBusy				: BOOL;
	bDone				: BOOL;
	bError				: BOOL;
END_VAR
CASE eMode OF
	E_MachineMode.MANUAL:
//		RobotWarehouseMoveManual_Ctrl.bExecute := bExecute;
//		RobotWarehouseMoveManual_Ctrl.bReset := bReset;
//		RobotWarehouseMoveManual_Ctrl.bAbort := E_Stop;
//		RobotWarehouseMoveManual_Ctrl.bOccupied := bOccupied;
		
//		bBusy := RobotWarehouseMoveManual_Status.bBusy;
//		bDone := RobotWarehouseMoveManual_Status.bDone;
//		bError := RobotWarehouseMoveManual_Status.bError;
		
	E_MachineMode.AUTO:
//		RobotWarehouseMoveAuto_Ctrl.bExecute := bExecute;
//		RobotWarehouseMoveAuto_Ctrl.bReset := bReset;
//		RobotWarehouseMoveAuto_Ctrl.bAbort := E_Stop;
//		RobotWarehouseMoveAuto_Ctrl.bOccupied := bOccupied;
		
//		bBusy := RobotWarehouseMoveAuto_Status.bBusy;
//		bDone := RobotWarehouseMoveAuto_Status.bDone;
//		bError := RobotWarehouseMoveAuto_Status.bError;
END_CASE
END_METHOD

METHOD M_StartHoming
VAR_INPUT
END_VAR
fbStorageHoming.xExecute := TRUE;
END_METHOD

METHOD M_Starting
M_StateComplete();
END_METHOD

METHOD M_StartSlideA_FeedIn : BOOL
VAR_INPUT
END_VAR
AutoMode_PulloutConveyor_Intern.PullOutConveyorInfo.CommandType :=E_PullOutConveyorCommandType.SlideA_FeedIn_Ext;

AutoMode_PulloutConveyor_Intern.Command.Execute := TRUE;

M_StartSlideA_FeedIn := TRUE; // Method end
END_METHOD

METHOD M_StartSlideA_FeedOut : BOOL
VAR_INPUT
	ReverseTimeDelay : Time;
END_VAR
AutoMode_PulloutConveyor_Intern.PullOutConveyorInfo.CommandType :=E_PullOutConveyorCommandType.SlideA_FeedOut_Ext;
AutoMode_PulloutConveyor_Intern.PullOutConveyorInfo.ConveyorReverseTime :=ReverseTimeDelay;
AutoMode_PulloutConveyor_Intern.Command.Execute := TRUE;

M_StartSlideA_FeedOut := TRUE; // Method end
END_METHOD

METHOD M_StartSlideB_FeedIn : BOOL
VAR_INPUT
END_VAR
AutoMode_PulloutConveyor_Intern.PullOutConveyorInfo.CommandType :=E_PullOutConveyorCommandType.SlideB_FeedIn_Ext;

AutoMode_PulloutConveyor_Intern.Command.Execute := TRUE;

M_StartSlideB_FeedIn := TRUE; // Method end
END_METHOD

METHOD M_StartSlideB_FeedOut : BOOL
VAR_INPUT
	ReverseTimeDelay : Time;
END_VAR
AutoMode_PulloutConveyor_Intern.PullOutConveyorInfo.CommandType :=E_PullOutConveyorCommandType.SlideB_FeedOut_Ext;
AutoMode_PulloutConveyor_Intern.PullOutConveyorInfo.ConveyorReverseTime :=ReverseTimeDelay;
AutoMode_PulloutConveyor_Intern.Command.Execute := TRUE;

M_StartSlideB_FeedOut := TRUE; // Method end
END_METHOD

METHOD M_StopHoming
VAR_INPUT
END_VAR
fbStorageHoming.xExecute := False;
END_METHOD

METHOD M_Stopped
//fbRobotRegionMove_BufferArea.Stop := FALSE;
M_StateComplete();
END_METHOD

METHOD M_Stopping

M_StateComplete();
END_METHOD

METHOD M_Suspended
M_StateComplete();
END_METHOD

METHOD M_Suspending
M_StateComplete();
END_METHOD

METHOD M_Undefined
M_StateComplete();
END_METHOD

METHOD M_Unholding
//fbRobotRegionMove_BufferArea.Stop := FALSE;
M_StateComplete();
END_METHOD

METHOD M_Unsuspending
M_StateComplete();
END_METHOD

END_FUNCTION_BLOCK

// ---- Library/20_MachineUnits/21_StorageArea/Service_Robot/FB_FeedInEmptyBoxWithRobot_V4.TcPOU
FUNCTION_BLOCK FB_FeedInEmptyBoxWithRobot_V4 EXTENDS FB_ObjectBase_V2 IMPLEMENTS IBasicElement
VAR_INPUT
    // Below are the components being controlled.
    Robot           : REFERENCE TO FB_FanucRobot_Basic_V2; // Fanuc Robot
    PullOutConveyor : REFERENCE TO FB_PullOutConveyorAction; // Allocated area pull out conveyor
    DiffSizeCV  	: REFERENCE TO FB_Motor; // Allocated area feed in conveyor(diff and same size conveyor)
	SameSizeCV 		: REFERENCE TO FB_Motor;
    WareHouse       : REFERENCE TO FB_WareHouse; // Storage area warehouse A and warehouse B conveyor and sensor
    //SameSizeFullSensor : REFERENCE TO BOOL; 				 // Because the same size sensor implement FB_ConveyorSameSize, so use reference to connect it
    Info  			: ST_FeedInEmptyBox_Info; // Setting the feedin emptybox action's parameter
    Input 			: REFERENCE TO ST_InputTable;
    Stop  			: BOOL;
END_VAR
VAR_OUTPUT
	AClampMoveDone	: BOOL;
	BClampMoveDone	: BOOL;
END_VAR
VAR
    tonPlaceSensorDelay    : TON;
    tonFeedInConveyorDelay : TON;
    tonTimeOut             : TON;
	bTimeOutIN			   : BOOL;
    tonFeedBoxTimeout      : TON;
	TON_WaitRobotClear	   : TON;
    strStatus              : STRING;
    _UniqueErrorCode       : STRING;
//    _Abort                 : BOOL;
    uiResumeStep           : UDINT;
	uiResumePlaceBothStep  : UINT;
	uiResumePlaceSingleStep: UINT;
    PreviousStrStatus      : STRING;
    PreviousErrorCode      : STRING;
	
	WorkingConveyor			: REFERENCE TO FB_Motor;
	SelectedSensor			: BOOL;
	bWorkingConveyorMoveForward : BOOL;
	bWorkingConveyorMoveBackward : BOOL;
	
	uiPickUpBothStep            : UDINT;
    uiPlaceBothStep             : UINT;
	uiPlaceSingleStep			: UINT;
	
	// Clamp work
	_AClampDoingWork	: BOOL;
	_BClampDoingWork	: BOOL;
	
	uiResumePickUpBothStep : UDINT;
	
	_bRetry	: BOOL;

	// Safe Pause
	bPauseLatched : BOOL;
	uiPauseFromStep : UDINT;
END_VAR

SUPER^.A10_StateControl();
A00_BasicUnits();

(*============================================================
Create Date : 2025/12/01
Last Update	: 2025/12/01
Change Log  : 2025/11/24，send flag A clamp done and B clamp done for C# use to SQL // Owner : Gamin
			  2025/12/1 ，Create V3__ import Kinsus version to fix Singal Clamp doing 	//Owner : Gamin
			  2026/03/23，新增 V4版本，新增輸送帶續做後移動功能。
			  2026/04/02，修正 STATE_Error 狀態。
============================================================*)

ACTION A00_BasicUnits:
tonTimeOut(IN:= bTimeOutIN AND NOT THIS^.Stop, PT:=T#60S);
tonFeedBoxTimeout(PT:=T#15s);
tonPlaceSensorDelay();
tonFeedInConveyorDelay(PT:=T#500MS);
TON_WaitRobotClear(PT := T#5S);
END_ACTION

METHOD PRIVATE M_BothClampReleasedBox : BOOL
VAR_INPUT
END_VAR
M_BothClampReleasedBox := THIS^.M_ClampAReleasedBox() AND THIS^.M_ClampBReleasedBox();
END_METHOD

METHOD M_CheckCommand : BOOL
VAR_INPUT
END_VAR

VAR_INST
	CheckBehavior : BOOL; // True : Behavior is correct
	CheckWareHouseSetting : BOOL; // True : WareHouse setting is correct
	CheckPullOutConveyorSetting : BOOL; // True : PullOut Conveyor setting is correct
	CheckPickUpArea : BOOL; // True : PickUp Area is correct
	CheckPlaceArea : BOOL; // True : Place Area is correct
END_VAR
// Memory clear
CheckBehavior := FALSE;
CheckWareHouseSetting := TRUE;
CheckPullOutConveyorSetting := TRUE;
CheckPickUpArea := TRUE;
CheckPlaceArea := TRUE;

// Check command is correct
IF info.ClampA_Setting.Behavior = E_ClampWork.Work OR info.ClampB_Setting.Behavior = E_ClampWork.Work THEN
	CheckBehavior := TRUE;
ELSE
	CheckBehavior := FALSE;
	strStatus := 'No clamp selected to work';
END_IF

IF info.ClampA_Setting.Behavior = E_ClampWork.Work THEN
	IF info.ClampA_Setting.PickUpArea = E_FeedInEmptyBox_PickUpArea.Undefined THEN
		CheckPickUpArea := FALSE;
		strStatus := 'ClampA pickup area undefined';
	END_IF
	IF info.ClampA_Setting.PlaceArea = E_FeedInEmptyBox_PlaceArea.Undefine THEN
		CheckPlaceArea := FALSE;
		strStatus := 'ClampA place area undefined';
	END_IF
	IF info.ClampA_Setting.PickUpArea = E_FeedInEmptyBox_PickUpArea.PullOutConveyor AND
	   info.ClampA_Setting.PullOutConveyorSetting = E_PullOutConveyorAddress.Undefined THEN
		CheckPullOutConveyorSetting := FALSE;
		strStatus := 'ClampA pullout slide undefined';
	END_IF
END_IF

IF info.ClampB_Setting.Behavior = E_ClampWork.Work THEN
	IF info.ClampB_Setting.PickUpArea = E_FeedInEmptyBox_PickUpArea.Undefined THEN
		CheckPickUpArea := FALSE;
		strStatus := 'ClampB pickup area undefined';
	END_IF
	IF info.ClampB_Setting.PlaceArea = E_FeedInEmptyBox_PlaceArea.Undefine THEN
		CheckPlaceArea := FALSE;
		strStatus := 'ClampB place area undefined';
	END_IF
	IF info.ClampB_Setting.PickUpArea = E_FeedInEmptyBox_PickUpArea.PullOutConveyor AND
	   info.ClampB_Setting.PullOutConveyorSetting = E_PullOutConveyorAddress.Undefined THEN
		CheckPullOutConveyorSetting := FALSE;
		strStatus := 'ClampB pullout slide undefined';
	END_IF
END_IF

M_CheckCommand := CheckBehavior AND CheckWareHouseSetting AND CheckPullOutConveyorSetting AND CheckPickUpArea AND CheckPlaceArea;

IF NOT (CheckBehavior AND CheckWareHouseSetting AND CheckPullOutConveyorSetting AND CheckPickUpArea AND CheckPlaceArea) THEN
	Status := strStatus;
	_Error := TRUE;
END_IF
END_METHOD

METHOD M_CheckUnitsNotBusy : BOOL
VAR_INPUT
END_VAR
M_CheckUnitsNotBusy := true; // need add units check
END_METHOD

METHOD M_CheckUnitsReady : BOOL
VAR_INPUT
END_VAR
M_CheckUnitsReady := NOT (Robot.Error (*OR PullOutConveyor.Error OR FeedInConveyor.bError OR WareHouse.bError*));
END_METHOD

METHOD PRIVATE M_ClampAReleasedBox : BOOL
VAR_INPUT
END_VAR
M_ClampAReleasedBox := NOT Robot._DI1.ClampA_Sensor AND Robot._DI1.ClampA_Open;
END_METHOD

METHOD PRIVATE M_ClampBReleasedBox : BOOL
VAR_INPUT
END_VAR
M_ClampBReleasedBox := NOT Robot._DI1.ClampB_Sensor AND Robot._DI1.ClampB_Open;
END_METHOD

METHOD PRIVATE M_HasBothClampBox : BOOL
VAR_INPUT
END_VAR
M_HasBothClampBox := THIS^.M_HasClampABox() AND THIS^.M_HasClampBBox();
END_METHOD

METHOD PRIVATE M_HasClampABox : BOOL
VAR_INPUT
END_VAR
M_HasClampABox := Robot._DI1.ClampA_Sensor AND NOT Robot._DI1.ClampA_Open;
END_METHOD

METHOD PRIVATE M_HasClampBBox : BOOL
VAR_INPUT
END_VAR
M_HasClampBBox := Robot._DI1.ClampB_Sensor AND NOT Robot._DI1.ClampB_Open;
END_METHOD

METHOD M_ReloadPulloutConveyorBox : BOOL
VAR_INPUT
	Execute : BOOL;
	SlideSelect : E_PullOutConveyorPosition;
END_VAR
VAR_INST
	uiReloadPulloutConveyorBoxStep : UDINT;
	fbExecute_Rtrig : R_TRIG;
	fbExecute_Ftrig : F_TRIG;
END_VAR
fbExecute_Rtrig(CLK := Execute);
fbExecute_Ftrig(CLK := Execute);
IF fbExecute_Rtrig.Q THEN
	uiReloadPulloutConveyorBoxStep := 100;
ELSIF fbExecute_Ftrig.Q THEN
	uiReloadPulloutConveyorBoxStep := 99000;
END_IF
CASE uiReloadPulloutConveyorBoxStep OF
	0 : 
		// Wait command
	99000:
//		PullOutConveyor.FixCylinderA1.M_MoveBackward('');
//		PullOutConveyor.FixCylinderA2.M_MoveBackward('');
//		PullOutConveyor.FixCylinderB1.M_MoveBackward('');
//		PullOutConveyor.FixCylinderB2.M_MoveBackward('');
END_CASE
END_METHOD

METHOD M_SelectActionMode : E_FeedInAction
VAR_INPUT
END_VAR
IF info.ClampA_Setting.Behavior = E_ClampWork.Work AND info.ClampB_Setting.Behavior <> E_ClampWork.Work THEN
	IF info.ClampA_Setting.PickUpArea = E_FeedInEmptyBox_PickUpArea.WareHouseA THEN
		M_SelectActionMode := E_FeedInAction.ClampA_WareHouseA;
	ELSIF info.ClampA_Setting.PickUpArea = E_FeedInEmptyBox_PickUpArea.WareHouseB THEN
		M_SelectActionMode := E_FeedInAction.ClampA_WareHouseB;
	ELSIF info.ClampA_Setting.PickUpArea = E_FeedInEmptyBox_PickUpArea.PullOutConveyor THEN
		M_SelectActionMode := E_FeedInAction.ClampA_PullOutConveyor;
	END_IF
ELSIF info.ClampA_Setting.Behavior <> E_ClampWork.Work AND info.ClampB_Setting.Behavior = E_ClampWork.Work THEN
	IF info.ClampB_Setting.PickUpArea = E_FeedInEmptyBox_PickUpArea.WareHouseA THEN
		M_SelectActionMode := E_FeedInAction.ClampB_WareHouseA;
	ELSIF info.ClampB_Setting.PickUpArea = E_FeedInEmptyBox_PickUpArea.WareHouseB THEN
		M_SelectActionMode := E_FeedInAction.ClampB_WareHouseB;
	ELSIF info.ClampB_Setting.PickUpArea = E_FeedInEmptyBox_PickUpArea.PullOutConveyor THEN
		M_SelectActionMode := E_FeedInAction.ClampB_PullOutConveyor;
	END_IF
ELSIF info.ClampA_Setting.Behavior = E_ClampWork.Work AND info.ClampB_Setting.Behavior = E_ClampWork.Work THEN
	IF info.ClampA_Setting.PickUpArea = E_FeedInEmptyBox_PickUpArea.PullOutConveyor THEN
		IF  info.ClampB_Setting.PickUpArea = E_FeedInEmptyBox_PickUpArea.WareHouseA THEN
			M_SelectActionMode := E_FeedInAction.A_PullOut_B_WareHouseA;
		ELSIF info.ClampB_Setting.PickUpArea = E_FeedInEmptyBox_PickUpArea.WareHouseB THEN
			M_SelectActionMode := E_FeedInAction.A_PullOut_B_WareHouseB;
		ELSIF info.ClampB_Setting.PickUpArea = E_FeedInEmptyBox_PickUpArea.PullOutConveyor THEN
			M_SelectActionMode := E_FeedInAction.A_PullOut_B_PullOut;
		END_IF
	ELSIF info.ClampA_Setting.PickUpArea = E_FeedInEmptyBox_PickUpArea.WareHouseA THEN
		IF info.ClampB_Setting.PickUpArea = E_FeedInEmptyBox_PickUpArea.WareHouseA THEN
			M_SelectActionMode := E_FeedInAction.A_WareHouseA_B_WareHouseA;
		ELSIF info.ClampB_Setting.PickUpArea = E_FeedInEmptyBox_PickUpArea.WareHouseB THEN
			M_SelectActionMode := E_FeedInAction.A_WareHouseA_B_WareHouseB;
		ELSIF info.ClampB_Setting.PickUpArea = E_FeedInEmptyBox_PickUpArea.PullOutConveyor THEN
			M_SelectActionMode := E_FeedInAction.A_WareHouseA_B_PullOut;
		END_IF
	ELSIF info.ClampA_Setting.PickUpArea = E_FeedInEmptyBox_PickUpArea.WareHouseB THEN
		IF info.ClampB_Setting.PickUpArea = E_FeedInEmptyBox_PickUpArea.WareHouseA THEN
			M_SelectActionMode := E_FeedInAction.A_WareHouseB_B_WareHouseA;
		ELSIF info.ClampB_Setting.PickUpArea = E_FeedInEmptyBox_PickUpArea.WareHouseB THEN
			M_SelectActionMode := E_FeedInAction.A_WareHouseB_B_WareHouseB;
		ELSIF info.ClampB_Setting.PickUpArea = E_FeedInEmptyBox_PickUpArea.PullOutConveyor THEN
			M_SelectActionMode := E_FeedInAction.A_WareHouseB_B_PullOut;
		END_IF
	END_IF
END_IF
END_METHOD

METHOD  M_STATE_ABORTED
VAR_INPUT
END_VAR
IF NOT _bRetry THEN
	Busy    := FALSE;
	Aborted := TRUE;
	Error   := TRUE;
	Status := strStatus ;
	UniqueErrorCode := _UniqueErrorCode;
	uiAbortingStep 		:= 0;
	_AbortCompleted 	:= FALSE;
	bTimeOutIN := FALSE;
END_IF

IF reset THEN
	_bRetry := TRUE;
	Error := _Error := FALSE;
	Abort := _Abort := Aborted := FALSE;
END_IF

IF NOT Execute THEN
    eState := STATE_RESETTING;
ELSIF Execute AND _bRetry AND NOT Robot._DI1.Error AND NOT Robot.Halt THEN
	Status := '';

	uiExecutingStep   := uiResumeStep;
	uiPlaceBothStep   := uiResumePlaceBothStep;
	uiPlaceSingleStep := uiResumePlaceSingleStep;
	uiPickUpBothStep  := uiResumePickUpBothStep;

	PreviousStrStatus := strStatus;
	PreviousErrorCode := _UniqueErrorCode;
	IF GVL_ADS.MachineState <>E_MachineState.Error THEN
		eSTATE:=STATE_EXECUTING;
	END_IF
END_IF
END_METHOD

METHOD  M_STATE_ABORTING
VAR_INPUT
END_VAR

CASE uiAbortingStep OF 
	0:
			_Abort 			:= FALSE;
			bTimeOutIN		:= FALSE;
			TON_WaitRobotClear.IN := false;
			_bRetry			  := FALSE;
			bWorkingConveyorMoveForward  := FALSE;
			bWorkingConveyorMoveBackward := FALSE;
			IF __ISVALIDREF(WorkingConveyor) THEN
				WorkingConveyor.M_MotorStop();
			END_IF
			WareHouse.M_ResetFeedInBox();
			WareHouse.M_ResetReloadBox();

			// 清除 Robot DO handshake 和周邊狀態（不管 Robot 是 Error 還是 Held）
			(* 
				comment edited By Gamin ，
				1. 續做不能清除手臂命令，如果是做雙爪夾盒，A爪做完B爪報錯進入到續做流程，如果在此清除掉手臂命令
					，後續回到executing 動作，此時的情境為A 已做完已夾完盒，等同於給手臂重新做的命令，，會有危險，
				2. 在Service 執行期間進入到錯誤狀態也不能清除圓帶的使用權，以免被其他的Serivce 搶走，會有危險
				3.  A、B done 不能清除，這旗標也可算是代表手臂該爪的動作完成，
				   如果A爪完成，B爪報錯，續做只接續著做B爪，這樣Service 結束就只會有B done。
			*)
//			Robot.M_ResetAllCommand();
//			Robot.Bzone_AllowWork := FALSE;
//			DiffSizeCV.M_MotorStop();
//			SameSizeCV.M_MotorStop();
//			DAS_CoreSys.MachineControl.fballocatearea.M_ReleasePulloutAccess(ControlAccess := E_RoundBeltControlAccess.FanucRobot);
//			AClampMoveDone	 := FALSE;
//			BClampMoveDone	 := FALSE;
//			_AClampDoingWork := FALSE;
//			_BClampDoingWork := FALSE;

			IF uiResumeStep = 99100 THEN
				uiAbortingStep := 5;
			ELSE
				uiAbortingStep := 10;
			END_IF
			
	5:		// only allow reset all command for 99100 retry path
			IF Robot.M_ResetAllCommand() THEN
				uiAbortingStep := 10;
			END_IF
			
	10:		// Stop PullOut conveyor for all steps that use it
			
			IF uiResumeStep = 38000 THEN
				CASE uiResumePickUpBothStep OF
					0,20:
							DAS_CoreSys.MachineControl.fballocatearea.M_StopStoragePulloutAction();
							uiAbortingStep := 50;
					10,99:
							uiAbortingStep := 50;
				END_CASE
			ELSIF uiResumeStep = 12000 OR uiResumeStep = 22000 OR
				  uiResumeStep = 32100 OR uiResumeStep = 35100 OR
				  uiResumeStep = 36000 OR uiResumeStep = 37000 THEN
				DAS_CoreSys.MachineControl.fballocatearea.M_StopStoragePulloutAction();
				uiAbortingStep := 100;
			ELSE
					uiAbortingStep := 50;
			END_IF
			
	50:		// 判別可以續做的子步驟，只給予這些子步驟 續做步驟，避免其他步驟回Executing 後，進入錯的子步驟
			IF uiResumeStep = 81000 THEN
				CASE uiPlaceBothStep OF
					30,40,50,90,99:
								uiPlaceBothStep	:= uiResumePlaceBothStep;
				ELSE
					;
				END_CASE
				uiAbortingStep	:= 100;
				
			ELSIF uiResumeStep = 61000 THEN
				CASE uiPlaceSingleStep OF
					400:
							uiPlaceSingleStep := uiResumePlaceSingleStep;
				ELSE
					;
				END_CASE
				uiAbortingStep := 100;
				
			ELSIF uiResumeStep = 71000 THEN
				CASE uiPlaceSingleStep OF 
					400:
							uiPlaceSingleStep := uiResumePlaceSingleStep;
				ELSE
					;
				END_CASE
				uiAbortingStep := 100;
				
			ELSE
				uiAbortingStep := 100;
			END_IF
			
	100:
			IF Robot._DI1.Error (*AND Robot.ErrMsg ='Laser detected'*)THEN
				uiAbortingStep := 200;
			ELSE
				uiAbortingStep := 9999;
			END_IF
	200:		
			 IF DAS_CoreSys.MachineControl.M_RobotResetCmd() THEN
				 uiAbortingStep := 300;
			 END_IF
	300:
			IF DAS_CoreSys.MachineControl.M_RobotStartCmd() THEN
				 uiAbortingStep := 400;
			 END_IF 
	400:
			IF Robot._DI1.Error THEN
		 		uiAbortingStep := 200;
			ELSE
				uiAbortingStep := 9999;
			END_IF
	9999:
			_AbortCompleted := TRUE;
	
END_CASE
IF strStatus = PreviousStrStatus THEN
	_UniqueErrorCode :=PreviousErrorCode;
END_IF
IF _AbortCompleted THEN
    eState := STATE_Aborted;
END_IF
END_METHOD

METHOD  M_STATE_DONE
VAR_INPUT
END_VAR
Busy   := FALSE;
_Error := Error := FALSE;
_Abort := Abort := FALSE;
Done   := TRUE;

IF NOT Execute THEN
    eState := STATE_RESETTING;
END_IF
END_METHOD

METHOD  M_STATE_DORMANT
VAR_INPUT
END_VAR
// Clear FB output
Busy            := FALSE;
Done            := FALSE;
Aborted         := FALSE;
Error           :=  FALSE;
ErrorID         := 0;
Status          := '';
_ResetCompleted := FALSE;
_Error          := FALSE;
_Executed       := FALSE;
uiExecutingStep := 0;
uiResettingStep := 0;
uiResumeStep			:= 0;
uiResumePickUpBothStep	:= 0;
uiResumePlaceBothStep	:= 0;
uiResumePlaceSingleStep	:= 0;
uiPickUpBothStep        := 0;
uiPlaceBothStep         := 0;
uiPlaceSingleStep		:= 0;

TON_WaitRobotClear.IN := false;
tonPlaceSensorDelay.IN :=FALSE;
tonFeedInConveyorDelay.IN :=FALSE;
bWorkingConveyorMoveForward  :=FALSE;
bWorkingConveyorMoveBackward :=FALSE;
AClampMoveDone	:= FALSE;
BClampMoveDone	:= FALSE;
_AClampDoingWork	:= FALSE;
_BClampDoingWork	:= FALSE;
bTimeOutIN 			:= FALSE;
_UniqueErrorCode 	:= '0';
PreviousStrStatus	:= '';
PreviousErrorCode	:= '';
tonPlaceSensorDelay.PT:=T#1.5S;
_AbortCompleted		:= FALSE;
_bRetry	:= FALSE;
Paused := FALSE;
bPauseLatched := FALSE;
uiPauseFromStep := 0;
//DAS.fbStorageArea.M_InactivePulloutConveyorInternCtrl();
// Wait Execute command

IF Execute AND NOT Stop THEN
    eState := STATE_EXECUTING;
END_IF
END_METHOD

METHOD  M_STATE_ERROR
VAR_INPUT
END_VAR
Robot.Bzone_AllowWork	:=FALSE;
Error 					:= TRUE;
Busy					:= FALSE;
status 					:= strStatus;

DAS_CoreSys.MachineControl.fballocatearea.M_StopStoragePulloutAction();
WareHouse.M_ResetFeedInBox();
WareHouse.M_ResetReloadBox();
DiffSizeCV.M_MotorStop();
SameSizeCV.M_MotorStop();

IF NOT Execute THEN
    eState := STATE_RESETTING;
END_IF
END_METHOD

METHOD M_STATE_EXECUTING
VAR_INPUT
END_VAR
VAR_INST
    ClampA_WareHouseCoordinates : ST_WareHouseCoordinates;
    ClampB_WareHouseCoordinates : ST_WareHouseCoordinates;

    BoxReady_1st                : BOOL;
    BoxReady_2nd                : BOOL;
    SlideClear_1st              : BOOL;
    SlideClear_2nd              : BOOL;
    TargetWarehouse             : E_WareHouse;
    DiffSizeSlide_Clear         : BOOL;
    SameSizeSlide_clear         : BOOL;
    ActionMode                  : E_FeedInAction;
END_VAR
VAR

END_VAR
// Set status busy
Busy := TRUE;
Robot.Bzone_AllowWork:=Robot._DI12.BzoneInWork;

IF __ISVALIDREF(WorkingConveyor) THEN
	IF 	bWorkingConveyorMoveForward AND NOT WorkingConveyor.InBackWard THEN
		WorkingConveyor.M_MoveForward();
	END_IF
	IF 	bWorkingConveyorMoveBackward AND NOT WorkingConveyor.InForWard THEN
		WorkingConveyor.M_MoveBackward();
	END_IF
END_IF


//Auto mode , just allow robot
IF THIS^.Stop THEN // Pending the timeout when Stop signal occur
	bTimeOutIN :=FALSE;
END_IF

CASE uiExecutingStep OF
    0:
	// 非自動模式直接報錯 (避免軸控衝突)
	IF GVL_Machine.PackTags[UnitNo.Storage].Status.UnitModeCurrent <> E_UnitMode.Auto THEN
		strStatus := 'Not in Auto mode';
		_UniqueErrorCode := 'E_NOT_AUTO_MODE';
		_Error := TRUE;
	ELSE
        // Clear variable
        ActionMode       := E_FeedInAction.Undefined;
        BoxReady_1st     := FALSE;
        BoxReady_2nd     := FALSE;
		bWorkingConveyorMoveForward  :=FALSE;
		bWorkingConveyorMoveBackward :=FALSE;

        uiPickUpBothStep := 0;
        uiPlaceBothStep  := 0;
		uiPlaceSingleStep := 0;
        // Check command
        IF M_CheckCommand() THEN
            uiExecutingStep := 10;
        END_IF
	END_IF
    10: // Start process, check units first
        IF M_CheckUnitsReady() THEN
            uiExecutingStep := 20;
        END_IF
    20: // Check units not busy state
        IF M_CheckUnitsNotBusy() THEN
            uiExecutingStep := 1000;
        END_IF
    1000:
        // Select action mode
        ActionMode      := M_SelectActionMode();
        uiExecutingStep := 1100;
    1100:
        // according action mode jump step
        CASE ActionMode OF
            E_FeedInAction.ClampA_WareHouseA:
                uiExecutingStep := 10000; // Go to start only ClampA pickup from WareHouseA
            E_FeedInAction.ClampA_WareHouseB:
                uiExecutingStep := 11000; // Go to Start only ClampA pickup from WareHouseB
            E_FeedInAction.ClampA_PullOutConveyor:
                uiExecutingStep := 12000; // Go to Start only ClampA pickup form PulloutConveyor
            E_FeedInAction.ClampB_WareHouseA:
                uiExecutingStep := 20000; // Go to Start only ClampB pickup from WareHouseA
            E_FeedInAction.ClampB_WareHouseB:
                uiExecutingStep := 21000; // Go to Start only ClampB pickup from WareHouseB
            E_FeedInAction.ClampB_PullOutConveyor:
                uiExecutingStep := 22000; // Go to Start only ClampB pickup from PulloutConveyor
            E_FeedInAction.A_WareHouseA_B_WareHouseA:
                uiExecutingStep := 30000; // Go to Start ClampA pickup from WarehouseA, ClampB pickup from WarehouseA
            E_FeedInAction.A_WareHouseA_B_WareHouseB:
                uiExecutingStep := 31000; // Go to Start ClampA pickup from WarehouseA, ClmapB pickup from WarehouseB
            E_FeedInAction.A_WareHouseA_B_PullOut:
                uiExecutingStep := 32000; // Go to Start ClampA pickup from WarehouseA, ClampB pickup from PulloutConveyor
            E_FeedInAction.A_WareHouseB_B_WareHouseA:
                uiExecutingStep := 33000; // Go to Start ClampA pickup from WarehouseB, ClampB pickup from WarehouseA
            E_FeedInAction.A_WareHouseB_B_WareHouseB:
                uiExecutingStep := 34000; // Go to Start ClampA pickup from WarehouseB, CLampB pickup from WarehouseB
            E_FeedInAction.A_WareHouseB_B_PullOut:
                uiExecutingStep := 35000; // Go to Start ClampA pickup from WarehouseB, ClampB pickup from PulloutConveyor
            E_FeedInAction.A_PullOut_B_WareHouseA:
                uiExecutingStep := 36000; // Go to Start ClampA pickup from PulloutConveyor, ClampB pickup from WarehouseA
            E_FeedInAction.A_PullOut_B_WareHouseB:
                uiExecutingStep := 37000; // Go to Start ClampA pickup from PulloutConveyor, ClampB pickup from WarehouseB
            E_FeedInAction.A_PullOut_B_PullOut:
                uiExecutingStep := 38000; // Go to Start ClampBoth pickup from PulloutConveyor
		ELSE
			strStatus := 'FeedInEmptyBox action mode undefined';
			Status := strStatus;
			_Error := TRUE;
        END_CASE
    10000: // Only clampA pickup box from WareHouseA
		bTimeOutIN :=TRUE;	
        IF NOT Robot._DI1.Done THEN
            ClampA_WareHouseCoordinates := info.ClampA_Setting.WareHouseSetting;
            WareHouse.M_StartReloadBox(WareHouseSelect := E_WareHouse.WareHouseA, WarehouseCoordinates := ClampA_WareHouseCoordinates);

            IF WareHouse.bReloadBox_Completed THEN
                BoxReady_1st 	 := TRUE;
				_AClampDoingWork := TRUE;
            END_IF

            Robot.M_StartWareHousePickUpBox_ClampA(WareHouseSelect := E_WareHouse.WareHouseA,
                                                   Info            := ClampA_WareHouseCoordinates,
                                                   BoxReady_1st    := BoxReady_1st);
												   
			//  robot doing AClamp done
			IF _AClampDoingWork AND THIS^.M_HasClampABox() THEN
				AClampMoveDone := TRUE;
			END_IF
        ELSE
            IF Robot.M_ResetWareHousePickUpBox_ClampA() THEN
				bTimeOutIN:=FALSE;
				IF THIS^.M_HasClampABox() THEN
                	uiExecutingStep := 60000; // only place clampA
				ELSE
					_Abort :=TRUE;
					uiResumeStep:=10000;
					strStatus := M_FormatManagedStatus(
						AlarmId := GVL_ErrorCode.GC_ALARM_STO_FEEDIN_EMPTY,
						InnerMessage := GVL_ErrorCode.GC_MSG_0120);
				END_IF
            END_IF
        END_IF
			
		IF tonTimeOut.Q THEN
			bTimeOutIN:=FALSE;
			uiResumeStep:=10000;
			_Abort :=TRUE;
			strStatus := M_FormatManagedStatus(
				AlarmId := GVL_ErrorCode.GC_ALARM_STO_FEEDIN_EMPTY,
				InnerMessage := GVL_ErrorCode.GC_MSG_0096);
			Status := strStatus;
			Error := TRUE;
		END_IF
		
    11000: // Only ClampA pickup box from WareHouseB
		bTimeOutIN :=TRUE;
        IF NOT Robot._di1.Done THEN
            ClampA_WareHouseCoordinates := info.ClampA_Setting.WareHouseSetting;
            WareHouse.M_StartReloadBox(WareHouseSelect := E_WareHouse.WareHouseB, WarehouseCoordinates := ClampA_WareHouseCoordinates);

            IF WareHouse.bReloadBox_Completed THEN
                BoxReady_1st 	 := TRUE;
				_AClampDoingWork := TRUE;
            END_IF

            Robot.M_StartWareHousePickUpBox_ClampA(WareHouseSelect := E_WareHouse.WareHouseB,
                                                   Info            := ClampA_WareHouseCoordinates,
                                                   BoxReady_1st    := BoxReady_1st);
			//  robot doing AClamp done
			IF _AClampDoingWork AND THIS^.M_HasClampABox() THEN
				AClampMoveDone := TRUE;
			END_IF
        ELSE
            IF Robot.M_ResetWareHousePickUpBox_ClampA() THEN
				bTimeOutIN:=FALSE;
				IF THIS^.M_HasClampABox() THEN
                	uiExecutingStep := 60000; // only place clampA
				ELSE
					_Abort 		:=TRUE;
					uiResumeStep:=11000;
					strStatus := M_FormatManagedStatus(	AlarmId := GVL_ErrorCode.GC_ALARM_STO_FEEDIN_EMPTY,
														InnerMessage := GVL_ErrorCode.GC_MSG_0120);
				END_IF
            END_IF
        END_IF

				
		IF tonTimeOut.Q THEN
			bTimeOutIN	:=FALSE;
			uiResumeStep:=11000;
			_Abort 		:=TRUE;
			strStatus := M_FormatManagedStatus(	AlarmId := GVL_ErrorCode.GC_ALARM_STO_FEEDIN_EMPTY,
												InnerMessage := GVL_ErrorCode.GC_MSG_0096);
			Status := strStatus;
			Error := TRUE;
		END_IF
		
    12000: // Only ClampA pickup box from pullout conveyor
		bTimeOutIN :=TRUE;	
        IF NOT Robot._di1.Done THEN
			DAS_CoreSys.MachineControl.fballocatearea.M_GetPulloutAccess(ControlAccess := E_RoundBeltControlAccess.FanucRobot);

            IF Info.ClampA_Setting.PullOutConveyorSetting = E_PullOutConveyorAddress.I3_Slide THEN
				DAS_CoreSys.MachineControl.fballocatearea.M_StartStoragePulloutAction(CommandType 	 := E_PullOutConveyorCommandType.SlideB_FeedIn_Ext,
																					 CV_BackwardTIme := T#0S,
																					 CV_ForwardTime  := T#0S);
																					 
            ELSIF Info.ClampA_Setting.PullOutConveyorSetting = E_PullOutConveyorAddress.I4_Slide THEN
				DAS_CoreSys.MachineControl.fballocatearea.M_StartStoragePulloutAction(CommandType 	 := E_PullOutConveyorCommandType.SlideA_FeedIn_Ext,
																					 CV_BackwardTIme := T#0S,
																					 CV_ForwardTime  := T#0S);
            ELSE
                strStatus := 'FB_FeedInEmptyBoxWithRobot_V3 ,Step 12000: Not define PulloutConveyor Slide';
				Status := strStatus;
                _Error := TRUE;
            END_IF
			
			IF DAS_CoreSys.MachineControl.fballocatearea.fbpulloutcv.Done THEN
					BoxReady_1st     := TRUE;
			END_IF
			
            Robot.M_StartPullOutConveyorPickUpBox_ClampA(ClampA_Address := Info.ClampA_Setting.PullOutConveyorSetting,
                                                         BoxReady       := BoxReady_1st);
        ELSE
            IF Robot.M_ResetPullOutConveyorPickUpBox_ClampA() THEN
                DAS_CoreSys.MachineControl.fbStorageArea.M_ResetSlideA_FeedIn();
				bTimeOutIN:=FALSE;
				IF THIS^.M_HasClampABox() THEN
                	uiExecutingStep := 60000; // only place clampA
				ELSE
					_Abort :=TRUE;
					uiResumeStep:=12000;
					strStatus := M_FormatManagedStatus(
						AlarmId := GVL_ErrorCode.GC_ALARM_STO_FEEDIN_EMPTY,
						InnerMessage := GVL_ErrorCode.GC_MSG_0120);
				END_IF
            END_IF
        END_IF;
				
		IF tonTimeOut.Q THEN
			bTimeOutIN:=FALSE;
			_Abort :=TRUE;
			uiResumeStep:=12000;
			strStatus := M_FormatManagedStatus(
				AlarmId := GVL_ErrorCode.GC_ALARM_STO_FEEDIN_EMPTY,
				InnerMessage := GVL_ErrorCode.GC_MSG_0096);
			Status := strStatus;
			Error := TRUE;
		END_IF
		
    20000: // Only clampB pickup box from WareHouseA
		bTimeOutIN :=TRUE;
        IF NOT Robot._di1.Done THEN
            ClampB_WareHouseCoordinates := info.ClampB_Setting.WareHouseSetting;
            WareHouse.M_StartReloadBox(WareHouseSelect := E_WareHouse.WareHouseA, WarehouseCoordinates := ClampB_WareHouseCoordinates);

            IF WareHouse.bReloadBox_Completed THEN
                BoxReady_2nd 	 := TRUE;
				_BClampDoingWork := TRUE;
            END_IF

            Robot.M_StartWareHousePickUpBox_ClampB(WareHouseSelect := E_WareHouse.WareHouseA,
                                                   Info            := ClampB_WareHouseCoordinates,
                                                   BoxReady_2nd    := BoxReady_2nd);
			// make sure robot doing Clamp done
			IF _BClampDoingWork AND THIS^.M_HasClampBBox() THEN
				BClampMoveDone := TRUE;
			END_IF
        ELSE
            IF Robot.M_ResetWareHousePickUpBox_ClampB() THEN
				bTimeOutIN:=FALSE;
				IF THIS^.M_HasClampBBox() THEN
                	uiExecutingStep := 70000; // only place clampA
				ELSE
					_Abort 		:= TRUE;
					uiResumeStep:= 20000;
					strStatus 	:= M_FormatManagedStatus( AlarmId := GVL_ErrorCode.GC_ALARM_STO_FEEDIN_EMPTY,
													  InnerMessage := GVL_ErrorCode.GC_MSG_0122);
				END_IF
            END_IF
        END_IF
					
		IF tonTimeOut.Q THEN
			bTimeOutIN	:= FALSE;
			_Abort 		:= TRUE;
			uiResumeStep:= 20000;
			strStatus 	:= M_FormatManagedStatus( AlarmId := GVL_ErrorCode.GC_ALARM_STO_FEEDIN_EMPTY,
												  InnerMessage := GVL_ErrorCode.GC_MSG_0096);
			Status 	:= strStatus;
			Error 	:= TRUE;
		END_IF
    21000: // Only ClampB pickup box from WareHouseB
		bTimeOutIN :=TRUE;	
        IF NOT Robot._di1.Done THEN
            ClampB_WareHouseCoordinates := info.ClampB_Setting.WareHouseSetting;
            WareHouse.M_StartReloadBox(WareHouseSelect := E_WareHouse.WareHouseB, WarehouseCoordinates := ClampB_WareHouseCoordinates);

            IF WareHouse.bReloadBox_Completed THEN
                BoxReady_2nd 	 := TRUE;
				_BClampDoingWork := TRUE;
            END_IF

            Robot.M_StartWareHousePickUpBox_ClampB(WareHouseSelect := E_WareHouse.WareHouseB,
                                                   Info            := ClampB_WareHouseCoordinates,
                                                   BoxReady_2nd    := BoxReady_2nd);
			// robot doing Clamp done
			IF _BClampDoingWork AND THIS^.M_HasClampBBox() THEN
				BClampMoveDone := TRUE;
			END_IF
        ELSE
            IF Robot.M_ResetWareHousePickUpBox_ClampB() THEN
				bTimeOutIN:=FALSE;
				IF THIS^.M_HasClampBBox() THEN
                	uiExecutingStep := 70000; // only place clampA
				ELSE
					_Abort 		:= TRUE;
					uiResumeStep:= 21000;
					strStatus 	:= M_FormatManagedStatus(AlarmId := GVL_ErrorCode.GC_ALARM_STO_FEEDIN_EMPTY,
													 InnerMessage := GVL_ErrorCode.GC_MSG_0122);
				END_IF
            END_IF
        END_IF
					
		IF tonTimeOut.Q THEN
			bTimeOutIN	:= FALSE;
			_Abort 		:= TRUE;
			uiResumeStep:= 21000;
			strStatus 	:= M_FormatManagedStatus(AlarmId := GVL_ErrorCode.GC_ALARM_STO_FEEDIN_EMPTY,
												 InnerMessage := GVL_ErrorCode.GC_MSG_0096);
			Status := strStatus;
			Error  := TRUE;
		END_IF

    22000: // Only ClampB pickup box from PullOut conveyor
		bTimeOutIN :=TRUE;	
        IF NOT Robot._di1.Done THEN
            DAS_CoreSys.MachineControl.fballocatearea.M_GetPulloutAccess(ControlAccess := E_RoundBeltControlAccess.FanucRobot);

            IF Info.ClampB_Setting.PullOutConveyorSetting = E_PullOutConveyorAddress.I3_Slide THEN
                DAS_CoreSys.MachineControl.fballocatearea.M_StartStoragePulloutAction(CommandType 	 := E_PullOutConveyorCommandType.SlideB_FeedIn_Ext,
																					 CV_BackwardTIme := T#0S,
																					 CV_ForwardTime  := T#0S);
            ELSIF Info.ClampB_Setting.PullOutConveyorSetting = E_PullOutConveyorAddress.I4_Slide THEN
                DAS_CoreSys.MachineControl.fballocatearea.M_StartStoragePulloutAction(CommandType 	 := E_PullOutConveyorCommandType.SlideA_FeedIn_Ext,
																					 CV_BackwardTIme := T#0S,
																					 CV_ForwardTime  := T#0S);
            ELSE
                strStatus := 'FB_FeedInEmptyBoxWithRobot_V3 ,Step 22000: Not define PulloutConveyor Slide';
				Status := strStatus;
                _Error := TRUE;
            END_IF
			
			IF DAS_CoreSys.MachineControl.fballocatearea.fbPulloutCV.Done THEN
				BoxReady_2nd := TRUE;
			END_IF
			
            Robot.M_StartPullOutConveyorPickUpBox_ClampB(ClampB_Address := Info.ClampB_Setting.PullOutConveyorSetting,
                                                         BoxReady       := BoxReady_2nd);
        ELSE
            IF Robot.M_ResetPullOutConveyorPickUpBox_ClampB() THEN
                DAS_CoreSys.MachineControl.fbStorageArea.M_ResetSlideA_FeedIn();
				bTimeOutIN:=FALSE;
				IF THIS^.M_HasClampBBox() THEN
                	uiExecutingStep := 70000; // only place clampA
				ELSE
					_Abort :=TRUE;
					uiResumeStep:=22000;
					strStatus := M_FormatManagedStatus(
						AlarmId := GVL_ErrorCode.GC_ALARM_STO_FEEDIN_EMPTY,
						InnerMessage := GVL_ErrorCode.GC_MSG_0122);
				END_IF
            END_IF
        END_IF;
				
		IF tonTimeOut.Q THEN
			bTimeOutIN:=FALSE;
			uiResumeStep:=22000;
			_Abort :=TRUE;
			strStatus := M_FormatManagedStatus(
				AlarmId := GVL_ErrorCode.GC_ALARM_STO_FEEDIN_EMPTY,
				InnerMessage := GVL_ErrorCode.GC_MSG_0096);
			Status := strStatus;
			Error := TRUE;
		END_IF
		
    30000: // ClampA pickup from WarehouseA, ClampB pickup from WarehouseA
        ClampA_WareHouseCoordinates := info.ClampA_Setting.WareHouseSetting;
        ClampB_WareHouseCoordinates := info.ClampB_Setting.WareHouseSetting;		
        CASE uiPickUpBothStep OF
            0: // ClampA target slide move the box to front side
                WareHouse.M_StartReloadBox(WareHouseSelect := E_WareHouse.WareHouseA, WarehouseCoordinates := ClampA_WareHouseCoordinates);

                IF WareHouse.bReloadBox_Completed THEN
                    BoxReady_1st     := TRUE;
					_AClampDoingWork := TRUE;
                    uiPickUpBothStep := 10;
                END_IF

            10: // wait Robot Allow continue
                IF Robot._DI1.Notification AND
                    NOT
                    WareHouse._stWarehouseList.ASide_Layers[ClampA_WareHouseCoordinates.Layer].stStatus.bSlides[ClampA_WareHouseCoordinates.Slide]
                    THEN
                    WareHouse.M_ResetReloadBox();

                    IF NOT WareHouse.bReloadBox_Completed THEN
                        uiPickUpBothStep := 20;
                    END_IF

                END_IF
            20: // ClampB target slide move the box to front slide
                WareHouse.M_StartReloadBox(WareHouseSelect := E_WareHouse.WareHouseA, WarehouseCoordinates := ClampB_WareHouseCoordinates);

                IF WareHouse.bReloadBox_Completed THEN
                    BoxReady_2nd     := TRUE;
					_BClampDoingWork := TRUE;
                    uiPickUpBothStep := 99;
                END_IF
            99:
        // wait reset
        END_CASE
			bTimeOutIN :=TRUE;	
        	Robot.M_StartWareHousePickUpBox_ClampBoth(WareHouseSelect := E_WareHouse.WareHouseA,
                                                  ClampA_Info     := ClampA_WareHouseCoordinates,
                                                  ClampB_Info     := ClampB_WareHouseCoordinates,
                                                  BoxReady_1st    := BoxReady_1st,
                                                  BoxReady_2nd    := BoxReady_2nd);
			// robot doing Clamp done
			IF _AClampDoingWork AND THIS^.M_HasClampABox() THEN
				AClampMoveDone := TRUE;
			END_IF						
			// robot doing Clamp done
			IF _BClampDoingWork AND THIS^.M_HasClampBBox() THEN
				BClampMoveDone := TRUE;
			END_IF

			IF Robot._DI1.Done THEN
				bTimeOutIN:=FALSE;
				IF THIS^.M_HasBothClampBox() THEN
					uiExecutingStep := 80000; // go to place step
				ELSE
					uiResumeStep:=30000;
					_Abort :=TRUE;
					strStatus := 'FB_FeedInEmptyBoxWithRobot_V4 Step 30000: both clamp pickup finished but clamp sensor not valid';
				END_IF
			END_IF
					
			IF tonTimeOut.Q THEN
				bTimeOutIN	:= FALSE;
				uiResumeStep:= 30000;
				_Abort 		:= TRUE;
				strStatus := M_FormatManagedStatus(
					AlarmId := GVL_ErrorCode.GC_ALARM_STO_FEEDIN_EMPTY,
					InnerMessage := GVL_ErrorCode.GC_MSG_0096);
				Status := strStatus;
				Error := TRUE;
			END_IF
		
    31000: // ClampA pickup from WarehouseA, ClampB pickup from WarehouseB
		bTimeOutIN :=TRUE;	
        IF NOT Robot._DI1.Done THEN
            ClampA_WareHouseCoordinates := info.ClampA_Setting.WareHouseSetting;
            WareHouse.M_StartReloadBox(WareHouseSelect := E_WareHouse.WareHouseA, WarehouseCoordinates := ClampA_WareHouseCoordinates);

            IF WareHouse.bReloadBox_Completed THEN
                BoxReady_1st 	 := TRUE;
				_AClampDoingWork := TRUE;
            END_IF

            Robot.M_StartWareHousePickUpBox_ClampA(WareHouseSelect := E_WareHouse.WareHouseA,
                                                   Info            := ClampA_WareHouseCoordinates,
                                                   BoxReady_1st    := BoxReady_1st);
												   
			// robot doing Clamp done
			IF _AClampDoingWork AND THIS^.M_HasClampABox() THEN
				AClampMoveDone := TRUE;
			END_IF
        ELSE
			bTimeOutIN:=FALSE;
			IF THIS^.M_HasClampABox() THEN
				uiExecutingStep := 31080;
			ELSE
				uiResumeStep:=31000;
				_Abort :=TRUE;
				strStatus := M_FormatManagedStatus(
					AlarmId := GVL_ErrorCode.GC_ALARM_STO_FEEDIN_EMPTY,
					InnerMessage := GVL_ErrorCode.GC_MSG_0120);
			END_IF
		END_IF
				
		IF tonTimeOut.Q THEN
			bTimeOutIN	:= FALSE;
			uiResumeStep:= 31000;
			_Abort 		:= TRUE;
			strStatus 	:= M_FormatManagedStatus(
				AlarmId := GVL_ErrorCode.GC_ALARM_STO_FEEDIN_EMPTY,
				InnerMessage := GVL_ErrorCode.GC_MSG_0096);
			Status := strStatus;
			Error  := TRUE;
		END_IF
		
	31080:
		Robot.M_ResetAllCommand(); // Clear command and go to place box
		IF NOT Robot._di1.Done THEN
			uiExecutingStep := 31100;// ClampA pickup finished, ClampB pickup start
		END_IF
		
    31100:
		bTimeOutIN :=TRUE;
        IF NOT Robot._di1.Done THEN
            ClampB_WareHouseCoordinates := info.ClampB_Setting.WareHouseSetting;
            WareHouse.M_StartReloadBox(WareHouseSelect := E_WareHouse.WareHouseB, WarehouseCoordinates := ClampB_WareHouseCoordinates);

            IF WareHouse.bReloadBox_Completed THEN
                BoxReady_2nd 	 := TRUE;
				_BClampDoingWork := TRUE;
            END_IF

            Robot.M_StartWareHousePickUpBox_ClampB(WareHouseSelect := E_WareHouse.WareHouseB,
                                                   Info            := ClampB_WareHouseCoordinates,
                                                   BoxReady_2nd    := BoxReady_2nd);
			
			// robot doing Clamp done
			IF _BClampDoingWork AND THIS^.M_HasClampBBox() THEN
				BClampMoveDone := TRUE;
			END_IF						   
												   
        ELSE
			bTimeOutIN:=FALSE;
			IF THIS^.M_HasClampBBox() THEN
				uiExecutingStep := 31180;
			ELSE
				uiResumeStep:=31100;
				_Abort :=TRUE;
				strStatus := M_FormatManagedStatus(
					AlarmId := GVL_ErrorCode.GC_ALARM_STO_FEEDIN_EMPTY,
					InnerMessage := GVL_ErrorCode.GC_MSG_0122);
			END_IF
		END_IF
					
		IF tonTimeOut.Q THEN
			bTimeOutIN	:= FALSE;
			uiResumeStep:= 31100;
			_Abort 		:= TRUE;
			strStatus 	:= M_FormatManagedStatus(
				AlarmId := GVL_ErrorCode.GC_ALARM_STO_FEEDIN_EMPTY,
				InnerMessage := GVL_ErrorCode.GC_MSG_0096);
			Status 	:= strStatus;
			Error 	:= TRUE;
		END_IF
		
	31180:
		Robot.M_ResetAllCommand(); // Clear command and go to place box
		IF NOT Robot._di1.Done THEN
			IF THIS^.M_HasBothClampBox() THEN
				uiExecutingStep := 80000;// ClampA pickup finished, ClampB pickup start
			ELSE
				uiResumeStep:=31100;
				_Abort :=TRUE;
				strStatus := 'FB_FeedInEmptyBoxWithRobot_V4 Step 31180: mixed pickup finished but both clamp sensor not valid';
			END_IF
		END_IF
		
    32000: // ClampA pickup from WarehouseA, ClampB pickup from PulloutConveyor
		bTimeOutIN :=TRUE;
        IF NOT Robot._DI1.Done THEN
            ClampA_WareHouseCoordinates := info.ClampA_Setting.WareHouseSetting;
            WareHouse.M_StartReloadBox(WareHouseSelect := E_WareHouse.WareHouseA, WarehouseCoordinates := ClampA_WareHouseCoordinates);

            IF WareHouse.bReloadBox_Completed THEN
                BoxReady_1st 	 := TRUE;
				_AClampDoingWork := TRUE;
            END_IF

            Robot.M_StartWareHousePickUpBox_ClampA(WareHouseSelect := E_WareHouse.WareHouseA,
                                                   Info            := ClampA_WareHouseCoordinates,
                                                   BoxReady_1st    := BoxReady_1st);
												   
			// robot doing Clamp done
			IF _AClampDoingWork AND THIS^.M_HasClampABox() THEN
				AClampMoveDone := TRUE;
			END_IF
			
        ELSE
			bTimeOutIN:=FALSE;
			IF THIS^.M_HasClampABox() THEN
				uiExecutingStep := 32080; // ClampA pickup finished, ClampB start	
			ELSE
				uiResumeStep:=32000;
				_Abort :=TRUE;
				strStatus := M_FormatManagedStatus(
					AlarmId := GVL_ErrorCode.GC_ALARM_STO_FEEDIN_EMPTY,
					InnerMessage := GVL_ErrorCode.GC_MSG_0120);
			END_IF
        END_IF
					
		IF tonTimeOut.Q THEN
			bTimeOutIN:=FALSE;
			uiResumeStep:=32000;
			_Abort :=TRUE;
			strStatus := M_FormatManagedStatus(
				AlarmId := GVL_ErrorCode.GC_ALARM_STO_FEEDIN_EMPTY,
				InnerMessage := GVL_ErrorCode.GC_MSG_0096);
			Status := strStatus;
			Error := TRUE;
		END_IF
	32080:
		Robot.M_ResetAllCommand();
		// Clear command and go to place box
		IF NOT Robot._di1.Done THEN
			uiExecutingStep := 32100;// ClampA pickup finished, ClampB start
		END_IF
    32100:
		bTimeOutIN :=TRUE;
        IF NOT Robot._di1.Done THEN
        DAS_CoreSys.MachineControl.fballocatearea.M_GetPulloutAccess(ControlAccess := E_RoundBeltControlAccess.FanucRobot);

            IF Info.ClampB_Setting.PullOutConveyorSetting = E_PullOutConveyorAddress.I3_Slide THEN
                        DAS_CoreSys.MachineControl.fballocatearea
                            .M_StartStoragePulloutAction(CommandType := E_PullOutConveyorCommandType.SlideB_FeedIn_Ext,
                                                         CV_BackwardTIme := T#0S,
                                                         CV_ForwardTime := T#0S);
            ELSIF Info.ClampB_Setting.PullOutConveyorSetting = E_PullOutConveyorAddress.I4_Slide THEN
                        DAS_CoreSys.MachineControl.fballocatearea
                            .M_StartStoragePulloutAction(CommandType := E_PullOutConveyorCommandType.SlideA_FeedIn_Ext,
                                                         CV_BackwardTIme := T#0S,
                                                         CV_ForwardTime := T#0S);
            ELSE
                strStatus := 'Not define PulloutConveyor Slide';
				Status := strStatus;
                _Error := TRUE;
            END_IF

            Robot.M_StartPullOutConveyorPickUpBox_ClampB(ClampB_Address := Info.ClampB_Setting.PullOutConveyorSetting,
                                                         BoxReady       := DAS_CoreSys.MachineControl.fballocatearea.fbPulloutCV.Done);
        ELSE
			bTimeOutIN:=FALSE;
			IF THIS^.M_HasClampBBox() THEN
				uiExecutingStep := 32180;
			ELSE
				uiResumeStep:=32100;
				_Abort :=TRUE;
				strStatus := M_FormatManagedStatus(
					AlarmId := GVL_ErrorCode.GC_ALARM_STO_FEEDIN_EMPTY,
					InnerMessage := GVL_ErrorCode.GC_MSG_0122);
			END_IF
		END_IF
					
		IF tonTimeOut.Q THEN
			bTimeOutIN:=FALSE;
			uiResumeStep:=32100;
			_Abort :=TRUE;
			strStatus := M_FormatManagedStatus(
				AlarmId := GVL_ErrorCode.GC_ALARM_STO_FEEDIN_EMPTY,
				InnerMessage := GVL_ErrorCode.GC_MSG_0096);
			Status := strStatus;
			Error := TRUE;
		END_IF
	32180:
		robot.M_ResetAllCommand();
		IF NOT Robot._DI1.Done THEN
			IF THIS^.M_HasBothClampBox() THEN
				uiExecutingStep := 80000;
			ELSE
				uiResumeStep:=32100;
				_Abort :=TRUE;
				strStatus := 'FB_FeedInEmptyBoxWithRobot_V4 Step 32180: mixed pickup finished but both clamp sensor not valid';
			END_IF
		END_IF
    33000: // ClampA Pickup from WarehouseB, ClampB pickup from WarehouseA
		bTimeOutIN :=TRUE;	
        IF NOT Robot._di1.Done THEN
            ClampA_WareHouseCoordinates := info.ClampA_Setting.WareHouseSetting;
            WareHouse.M_StartReloadBox(WareHouseSelect := E_WareHouse.WareHouseB, WarehouseCoordinates := ClampA_WareHouseCoordinates);

            IF WareHouse.bReloadBox_Completed THEN
                BoxReady_1st 	 := TRUE;
				_AClampDoingWork := TRUE;
            END_IF

            Robot.M_StartWareHousePickUpBox_ClampA(WareHouseSelect := E_WareHouse.WareHouseB,
                                                   Info            := ClampA_WareHouseCoordinates,
                                                   BoxReady_1st    := BoxReady_1st);
												   
			// robot doing Clamp done
			IF _AClampDoingWork AND THIS^.M_HasClampABox() THEN
				AClampMoveDone := TRUE;
			END_IF
			
        ELSE
			bTimeOutIN:=FALSE;
			IF THIS^.M_HasClampABox() THEN
				uiExecutingStep := 33080;
			ELSE
				uiResumeStep:=33000;
				_Abort :=TRUE;
				strStatus := M_FormatManagedStatus(
					AlarmId := GVL_ErrorCode.GC_ALARM_STO_FEEDIN_EMPTY,
					InnerMessage := GVL_ErrorCode.GC_MSG_0120);
			END_IF
		END_IF
					
		IF tonTimeOut.Q THEN
			bTimeOutIN:=FALSE;
			uiResumeStep:=33000;
			_Abort :=TRUE;
			strStatus := M_FormatManagedStatus(
				AlarmId := GVL_ErrorCode.GC_ALARM_STO_FEEDIN_EMPTY,
				InnerMessage := GVL_ErrorCode.GC_MSG_0096);
			Status := strStatus;
			Error := TRUE;
		END_IF
	33080:
		Robot.M_ResetAllCommand(); // Clear command and go to place box
		IF NOT Robot._DI1.Done THEN
                uiExecutingStep := 33100; // only place clampA
        END_IF
    
	33100:
		bTimeOutIN :=TRUE;
        IF NOT Robot._di1.Done THEN
            ClampB_WareHouseCoordinates := info.ClampB_Setting.WareHouseSetting;
            WareHouse.M_StartReloadBox(WareHouseSelect := E_WareHouse.WareHouseA, WarehouseCoordinates := ClampB_WareHouseCoordinates);

            IF WareHouse.bReloadBox_Completed THEN
                BoxReady_2nd 	 := TRUE;
				_BClampDoingWork := TRUE;
            END_IF

            Robot.M_StartWareHousePickUpBox_ClampB(WareHouseSelect := E_WareHouse.WareHouseA,
                                                   Info            := ClampB_WareHouseCoordinates,
                                                   BoxReady_2nd    := BoxReady_2nd);
			// robot doing Clamp done
			IF _BClampDoingWork AND THIS^.M_HasClampBBox() THEN
				BClampMoveDone := TRUE;
			END_IF										   									   
        ELSE
			IF THIS^.M_HasClampBBox() THEN
				Robot.M_ResetAllCommand(); // Clear command and go to place box
				IF NOT Robot._DI1.Done THEN
					bTimeOutIN:=FALSE;
					IF THIS^.M_HasBothClampBox() THEN
						uiExecutingStep := 80000; // only place clampA
					ELSE
						uiResumeStep:=33100;
						_Abort :=TRUE;
						strStatus := 'FB_FeedInEmptyBoxWithRobot_V4 Step 33100: mixed pickup finished but both clamp sensor not valid';
					END_IF
				END_IF
			ELSE
				bTimeOutIN:=FALSE;
				uiResumeStep:=33100;
				_Abort :=TRUE;
				strStatus := M_FormatManagedStatus(
					AlarmId := GVL_ErrorCode.GC_ALARM_STO_FEEDIN_EMPTY,
					InnerMessage := GVL_ErrorCode.GC_MSG_0122);
			END_IF
        END_IF
				
		IF tonTimeOut.Q THEN
			bTimeOutIN:=FALSE;
			uiResumeStep:=33100;
			_Abort :=TRUE;
			strStatus := M_FormatManagedStatus(
				AlarmId := GVL_ErrorCode.GC_ALARM_STO_FEEDIN_EMPTY,
				InnerMessage := GVL_ErrorCode.GC_MSG_0097);
			Status := strStatus;
			Error := TRUE;
		END_IF
		
    34000: // ClampA pickup from WarehouseB, ClampB pickup from WarehouseB
        ClampA_WareHouseCoordinates := info.ClampA_Setting.WareHouseSetting;
        ClampB_WareHouseCoordinates := info.ClampB_Setting.WareHouseSetting;

        CASE uiPickUpBothStep OF
            0: // ClampA target slide move the box to front side
                WareHouse.M_StartReloadBox(WareHouseSelect := E_WareHouse.WareHouseB, WarehouseCoordinates := ClampA_WareHouseCoordinates);

                IF WareHouse.bReloadBox_Completed THEN
                    BoxReady_1st     := TRUE;
					_AClampDoingWork := TRUE;
                    uiPickUpBothStep := 10;
                END_IF

            10: // wait Robot Allow continue
                IF Robot._DI1.Notification AND
                    NOT
                    WareHouse._stWarehouseList.BSide_Layers[ClampA_WareHouseCoordinates.Layer].stStatus.bSlides[ClampA_WareHouseCoordinates.Slide]
                    THEN
                    WareHouse.M_ResetReloadBox();

                    IF NOT WareHouse.bReloadBox_Completed THEN
                        uiPickUpBothStep := 20;
                    END_IF

                END_IF
            20: // ClampB target slide move the box to front slide
                WareHouse.M_StartReloadBox(WareHouseSelect := E_WareHouse.WareHouseB, WarehouseCoordinates := ClampB_WareHouseCoordinates);

                IF WareHouse.bReloadBox_Completed THEN
                    BoxReady_2nd     := TRUE;
					_BClampDoingWork := TRUE;
                    uiPickUpBothStep := 99;
                END_IF
            99:
        // wait reset
        END_CASE
		bTimeOutIN :=TRUE;
        Robot.M_StartWareHousePickUpBox_ClampBoth(WareHouseSelect := E_WareHouse.WareHouseB,
                                                  ClampA_Info     := ClampA_WareHouseCoordinates,
                                                  ClampB_Info     := ClampB_WareHouseCoordinates,
                                                  BoxReady_1st    := BoxReady_1st,
                                                  BoxReady_2nd    := BoxReady_2nd);
												  
		// robot doing Clamp done
		IF _BClampDoingWork AND THIS^.M_HasClampBBox() THEN
			BClampMoveDone := TRUE;
		END_IF	
		// robot doing Clamp done
		IF _AClampDoingWork AND THIS^.M_HasClampABox() THEN
			AClampMoveDone := TRUE;
		END_IF	

        IF Robot._DI1.Done THEN
			bTimeOutIN:=FALSE;
			IF THIS^.M_HasBothClampBox() THEN
            	uiExecutingStep := 80000; // go to place step
			ELSE
				uiResumeStep:=34000;
				_Abort :=TRUE;
				strStatus := 'FB_FeedInEmptyBoxWithRobot_V4 Step 34000: both clamp pickup finished but clamp sensor not valid';
			END_IF
        END_IF
		
					
		IF tonTimeOut.Q THEN
			bTimeOutIN:=FALSE;
			uiResumeStep:=34000;
			_Abort :=TRUE;
			strStatus := M_FormatManagedStatus(
				AlarmId := GVL_ErrorCode.GC_ALARM_STO_FEEDIN_EMPTY,
				InnerMessage := GVL_ErrorCode.GC_MSG_0096);
			Status := strStatus;
			Error := TRUE;
		END_IF
		
    35000: // ClampA pickup from WarehouseB, ClampB pickup from PulloutConveyor
		bTimeOutIN :=TRUE;		
		IF NOT Robot._DI1.Done THEN
            ClampA_WareHouseCoordinates := info.ClampA_Setting.WareHouseSetting;
            WareHouse.M_StartReloadBox(WareHouseSelect := E_WareHouse.WareHouseB, WarehouseCoordinates := ClampA_WareHouseCoordinates);

            IF WareHouse.bReloadBox_Completed THEN
                BoxReady_1st := TRUE;
				_AClampDoingWork := TRUE;
            END_IF

            Robot.M_StartWareHousePickUpBox_ClampA(WareHouseSelect := E_WareHouse.WareHouseA,
                                                   Info            := ClampA_WareHouseCoordinates,
                                                   BoxReady_1st    := BoxReady_1st);
			// robot doing Clamp done
				IF _AClampDoingWork AND THIS^.M_HasClampABox() THEN
					AClampMoveDone := TRUE;
				END_IF									   
        ELSE
		  tonTimeOut.IN:=FALSE;
		  IF THIS^.M_HasClampABox() THEN
		  	uiExecutingStep := 35100; // ClampA pickup finished, ClampB start 
		  ELSE
			uiResumeStep:=35000;
			_Abort :=TRUE;
			strStatus := M_FormatManagedStatus(
				AlarmId := GVL_ErrorCode.GC_ALARM_STO_FEEDIN_EMPTY,
				InnerMessage := GVL_ErrorCode.GC_MSG_0120);
		  END_IF
		END_IF
		  tonTimeOut.IN :=TRUE;   
		IF tonTimeOut.Q THEN
		  tonTimeOut.IN:=FALSE;
		  uiResumeStep:=35000;
		  _Abort :=TRUE;
		  strStatus := M_FormatManagedStatus(
		  	AlarmId := GVL_ErrorCode.GC_ALARM_STO_FEEDIN_EMPTY,
		  	InnerMessage := GVL_ErrorCode.GC_MSG_0096);
		  Status := strStatus;
		  Error := TRUE;
    	END_IF
		
    35100:
		bTimeOutIN :=TRUE;	
        IF NOT Robot._di1.Done THEN
        DAS_CoreSys.MachineControl.fballocatearea.M_GetPulloutAccess(ControlAccess := E_RoundBeltControlAccess.FanucRobot);

            IF Info.ClampB_Setting.PullOutConveyorSetting = E_PullOutConveyorAddress.I3_Slide THEN
                        DAS_CoreSys.MachineControl.fballocatearea
                            .M_StartStoragePulloutAction(CommandType := E_PullOutConveyorCommandType.SlideB_FeedIn_Ext,
                                                         CV_BackwardTIme := T#0S,
                                                         CV_ForwardTime := T#0S);
            ELSIF Info.ClampB_Setting.PullOutConveyorSetting = E_PullOutConveyorAddress.I4_Slide THEN
                        DAS_CoreSys.MachineControl.fballocatearea
                            .M_StartStoragePulloutAction(CommandType := E_PullOutConveyorCommandType.SlideA_FeedIn_Ext,
                                                         CV_BackwardTIme := T#0S,
                                                         CV_ForwardTime := T#0S);
            ELSE
                strStatus := 'Not define PulloutConveyor Slide';
				Status := strStatus;
                _Error := TRUE;
            END_IF

            Robot.M_StartPullOutConveyorPickUpBox_ClampB(ClampB_Address := Info.ClampB_Setting.PullOutConveyorSetting,
                                                         BoxReady       := DAS_CoreSys.MachineControl.fballocatearea.fbPulloutCV.Done);
        ELSE
            IF Robot.M_ResetPullOutConveyorPickUpBox_ClampB() THEN
            DAS_CoreSys.MachineControl.fballocatearea.M_StopStoragePulloutAction();
				bTimeOutIN:=FALSE;
				IF THIS^.M_HasClampBBox() AND THIS^.M_HasBothClampBox() THEN
                	uiExecutingStep := 80000; // only place clampA
				ELSE
					uiResumeStep:=35100;
					_Abort :=TRUE;
					strStatus := 'FB_FeedInEmptyBoxWithRobot_V4 Step 35100: mixed pickup finished but both clamp sensor not valid';
				END_IF
            END_IF
        END_IF;
					
		IF tonTimeOut.Q THEN
			bTimeOutIN:=FALSE;
			uiResumeStep:=35100;
			_Abort :=TRUE;
			strStatus := M_FormatManagedStatus(
				AlarmId := GVL_ErrorCode.GC_ALARM_STO_FEEDIN_EMPTY,
				InnerMessage := GVL_ErrorCode.GC_MSG_0096);
			Status := strStatus;
			Error := TRUE;
		END_IF
		
